(* If state methods are not disabled, run the stopped entry method. *)
IF NOT in_bDisableStateMethods THEN
	THIS^.M_LogMessage('Entered $'Stopped$' state.');
	THIS^.M110_Stopped_Entry();
ELSE
	THIS^.M_LogWarning('State methods disabled! Entered $'Stopped$' state. Waiting for transition...');
END_IF
END_ACTION

ACTION A111_Stopped:
{attribute 'hide'}
(* If state methods are not disabled, run the stopped method. *)
IF NOT in_bDisableStateMethods THEN
	THIS^.M111_Stopped(bReset => sm_bResetCmd, bAbort => sm_bAbortCmd);
	IF sm_bAbortCmd THEN
		sm_bAbort := TRUE;
	ELSIF sm_bResetCmd THEN
		sm_bReset := TRUE;
	END_IF
END_IF
END_ACTION

ACTION A112_Stopped_Exit:
{attribute 'hide'}
(* If state methods are not disabled, run the stopped exit method. *)
IF NOT in_bDisableStateMethods THEN
	THIS^.M112_Stopped_Exit();
END_IF
END_ACTION

{attribute 'hide'}
METHOD M110_Stopped_Entry : BOOL
END_METHOD

{attribute 'hide'}
METHOD M111_Stopped : BOOL
VAR_OUTPUT
	(* Move to the Resetting state*)
	bReset	: BOOL	:= FALSE;
	(* Move to the Aborting state*)
	bAbort	: BOOL	:= FALSE;
END_VAR
END_METHOD

{attribute 'hide'}
METHOD M112_Stopped_Exit : BOOL
END_METHOD

ACTION A200_Resetting_Entry:
{attribute 'hide'}
sm_enumState := E_PackMLState.Resetting;
sm_bIdle := FALSE;
sm_bStop := FALSE;

IF NOT in_bDisableStateMethods THEN
	THIS^.M_LogMessage('Entered $'Resetting$' state.');
	THIS^.M200_Resetting_Entry();
ELSE
	THIS^.M_LogWarning('State methods disabled! Entered $'Resetting$' state. Skipping to $'Idle$' state...');
	sm_bIdle := TRUE;
END_IF
END_ACTION

ACTION A201_Resetting:
{attribute 'hide'}
IF NOT in_bDisableStateMethods THEN
	THIS^.M201_Resetting(bIdle => sm_bIdleCmd, bStop => sm_bStopCmd, bAbort => sm_bAbortCmd);
	IF sm_bAbortCmd THEN
		sm_bAbort := TRUE;
	ELSIF sm_bStopCmd THEN
		sm_bStop := TRUE;
	ELSIF sm_bIdleCmd THEN
		sm_bIdle := TRUE;
	END_IF
END_IF
END_ACTION

ACTION A202_Resetting_Exit:
{attribute 'hide'}
IF NOT in_bDisableStateMethods THEN
	THIS^.M202_Resetting_Exit();
END_IF
END_ACTION

{attribute 'hide'}
METHOD M200_Resetting_Entry : BOOL
END_METHOD

{attribute 'hide'}
METHOD M201_Resetting : BOOL
VAR_OUTPUT
	(* Move to the Idle state*)
	bIdle	: BOOL	:= FALSE;
	(* Move to the Stopping state*)
	bStop	: BOOL	:= FALSE;
	(* Move to the Aborting state*)
	bAbort	: BOOL	:= FALSE;
END_VAR
// Move to idle state by default
bIdle := TRUE;
END_METHOD

{attribute 'hide'}
METHOD M202_Resetting_Exit : BOOL
END_METHOD

ACTION A210_Idle_Entry:
{attribute 'hide'}
sm_enumState := E_PackMLState.Idle;
sm_bStart := FALSE;

IF NOT in_bDisableStateMethods THEN
	THIS^.M_LogMessage('Entered $'Idle$' state.');
	THIS^.M210_Idle_Entry();
ELSE
	THIS^.M_LogWarning('State methods disabled! Entered $'Idle$' state. Waiting for transtion...');
END_IF
END_ACTION

ACTION A211_Idle:
{attribute 'hide'}
IF NOT in_bDisableStateMethods THEN
	THIS^.M211_Idle(bStart => sm_bStartCmd, bStop => sm_bStopCmd, bAbort => sm_bAbortCmd);
	IF sm_bAbortCmd THEN
		sm_bAbort := TRUE;
	ELSIF sm_bStopCmd THEN
		sm_bStop := TRUE;
	ELSIF sm_bStartCmd THEN
		sm_bStart := TRUE;
	END_IF
END_IF
END_ACTION

ACTION A212_Idle_Exit:
{attribute 'hide'}
IF NOT in_bDisableStateMethods THEN
	THIS^.M212_Idle_Exit();
END_IF
END_ACTION

{attribute 'hide'}
METHOD M210_Idle_Entry : BOOL
END_METHOD

{attribute 'hide'}
METHOD M211_Idle : BOOL
VAR_OUTPUT
	(* Move to the Starting state*)
	bStart	: BOOL	:= FALSE;
	(* Move to the Stopping state*)
	bStop	: BOOL	:= FALSE;
	(* Move to the Aborting state*)
	bAbort	: BOOL	:= FALSE;
END_VAR
END_METHOD

{attribute 'hide'}
METHOD M212_Idle_Exit : BOOL
END_METHOD

ACTION A300_Starting_Entry:
{attribute 'hide'}
sm_enumState := E_PackMLState.Starting;
sm_bStarted := FALSE;

IF NOT in_bDisableStateMethods THEN
	THIS^.M_LogMessage('Entered $'Starting$' state.');
	THIS^.M300_Starting_Entry();
ELSE
	THIS^.M_LogWarning('State methods disabled! Entered $'Starting$' state. Skipping to $'Execute$' state...');
	sm_bStarted := TRUE;
END_IF
END_ACTION

ACTION A301_Starting:
{attribute 'hide'}
IF NOT in_bDisableStateMethods THEN
	THIS^.M301_Starting(
		bStarted => sm_bStartedCmd,
		bStop => sm_bStopCmd,
		bAbort => sm_bAbortCmd);
	IF sm_bAbortCmd THEN
		sm_bAbort := TRUE;
	ELSIF sm_bStopCmd THEN
		sm_bStop := TRUE;
	ELSIF sm_bStartedCmd THEN
		sm_bStarted := TRUE;
	END_IF
END_IF
END_ACTION

ACTION A302_Starting_Exit:
{attribute 'hide'}
IF NOT in_bDisableStateMethods THEN
	THIS^.M302_Starting_Exit();
END_IF
END_ACTION

{attribute 'hide'}
METHOD M300_Starting_Entry : BOOL
END_METHOD

{attribute 'hide'}
METHOD M301_Starting : BOOL
VAR_OUTPUT
	(* Move to the Execute state*)
	bStarted	: BOOL	:= FALSE;
	(* Move to the Stopping state*)
	bStop		: BOOL	:= FALSE;
	(* Move to the Aborting state*)
	bAbort		: BOOL	:= FALSE;
END_VAR
// Move to execute state by default
bStarted := TRUE;
END_METHOD

{attribute 'hide'}
METHOD M302_Starting_Exit : BOOL
END_METHOD

ACTION A310_Execute_Entry:
{attribute 'hide'}
sm_enumState := E_PackMLState.Execute;
sm_bFinished := FALSE;
sm_bHold := FALSE;
sm_bSuspend := FALSE;

IF NOT in_bDisableStateMethods THEN
	THIS^.M_LogMessage('Entered $'Execute$' state.');
	THIS^.M310_Execute_Entry();
ELSE
	THIS^.M_LogWarning('State methods disabled! Entered $'Execute$' state. Waiting for transition...');
END_IF
END_ACTION

ACTION A311_Execute:
{attribute 'hide'}
IF NOT in_bDisableStateMethods THEN
	THIS^.M311_Execute(
		bFinished => sm_bFinishedCmd,
		bHold => sm_bHoldCmd,
		bSuspend => sm_bSuspendCmd,
		bStop => sm_bStopCmd,
		bAbort => sm_bAbortCmd);
	IF sm_bAbortCmd THEN
		sm_bAbort := TRUE;
	ELSIF sm_bStopCmd THEN
		sm_bStop := TRUE;
	ELSIF sm_bHoldCmd THEN
		sm_bHold := TRUE;
	ELSIF sm_bSuspendCmd THEN
		sm_bSuspend := TRUE;
	ELSIF sm_bFinishedCmd THEN
		sm_bFinished := TRUE;
	END_IF
END_IF
END_ACTION

ACTION A312_Execute_Exit:
{attribute 'hide'}
IF NOT in_bDisableStateMethods THEN
	THIS^.M312_Execute_Exit();
END_IF
END_ACTION

{attribute 'hide'}
METHOD M310_Execute_Entry : BOOL
END_METHOD

{attribute 'hide'}
METHOD M311_Execute : BOOL
VAR_OUTPUT
	(* Move to the Completing state*)
	bFinished	: BOOL	:= FALSE;
	(* Move to the Holding state*)
	bHold		: BOOL	:= FALSE;
	(* Move to the Suspending state*)
	bSuspend	: BOOL	:= FALSE;
	(* Move to the Stopping state*)
	bStop		: BOOL	:= FALSE;
	(* Move to the Aborting state*)
	bAbort		: BOOL	:= FALSE;
END_VAR
END_METHOD

{attribute 'hide'}
METHOD M312_Execute_Exit : BOOL
END_METHOD

ACTION A320_Completing_Entry:
{attribute 'hide'}
sm_enumState := E_PackMLState.Completing;
sm_bCompleted := FALSE;

IF NOT in_bDisableStateMethods THEN
	THIS^.M_LogMessage('Entered $'Completing$' state.');
	THIS^.M320_Completing_Entry();
ELSE
	THIS^.M_LogWarning('State methods disabled! Entered $'Completing$' state. Skipping to $'Completed$' state...');
	sm_bCompleted := TRUE;
END_IF
END_ACTION

ACTION A321_Completing:
{attribute 'hide'}
IF NOT in_bDisableStateMethods THEN
	THIS^.M321_Completing(
		bCompleted => sm_bCompletedCmd,
		bStop => sm_bStopCmd,
		bAbort => sm_bAbortCmd);
	IF sm_bAbortCmd THEN
		sm_bAbort := TRUE;
	ELSIF sm_bStopCmd THEN
		sm_bStop := TRUE;
	ELSIF sm_bCompletedCmd THEN
		sm_bCompleted := TRUE;
	END_IF
END_IF
END_ACTION

ACTION A322_Completing_Exit:
{attribute 'hide'}
IF NOT in_bDisableStateMethods THEN
	THIS^.M322_Completing_Exit();
END_IF
END_ACTION

{attribute 'hide'}
METHOD M320_Completing_Entry : BOOL
END_METHOD

{attribute 'hide'}
METHOD M321_Completing : BOOL
VAR_OUTPUT
	(* Move to the Complete state*)
	bCompleted	: BOOL	:= FALSE;
	(* Move to the Stopping state*)
	bStop		: BOOL	:= FALSE;
	(* Move to the Aborting state*)
	bAbort		: BOOL	:= FALSE;
END_VAR
// Move to complete state by default.
bCompleted := TRUE;
END_METHOD

{attribute 'hide'}
METHOD M322_Completing_Exit : BOOL
END_METHOD

ACTION A330_Complete_Entry:
{attribute 'hide'}
sm_enumState := E_PackMLState.Complete;
sm_bReturn := FALSE;

IF NOT in_bDisableStateMethods THEN
	THIS^.M_LogMessage('Entered $'Complete$' state.');
	THIS^.M330_Complete_Entry();
ELSE
	THIS^.M_LogWarning('State methods disabled! Entered $'Complete$' state. Waiting for transition...');
END_IF
END_ACTION

ACTION A331_Complete:
{attribute 'hide'}
IF NOT in_bDisableStateMethods THEN
	THIS^.M331_Complete(
		bReturn => sm_bReturnCmd,
		bStop => sm_bStopCmd,
		bAbort => sm_bAbortCmd);
	IF sm_bAbortCmd THEN
		sm_bAbort := TRUE;
	ELSIF sm_bStopCmd THEN
		sm_bStop := TRUE;
	ELSIF sm_bReturnCmd THEN
		sm_bReturn := TRUE;
	END_IF
END_IF
END_ACTION

ACTION A332_Complete_Exit:
{attribute 'hide'}
IF NOT in_bDisableStateMethods THEN
	THIS^.M332_Complete_Exit();
END_IF
END_ACTION

{attribute 'hide'}
METHOD M330_Complete_Entry : BOOL
END_METHOD

{attribute 'hide'}
METHOD M331_Complete : BOOL
VAR_OUTPUT
	(* Move to the Resetting state*)
	bReturn	: BOOL	:= FALSE;
	(* Move to the Stopping state*)
	bStop	: BOOL	:= FALSE;
	(* Move to the Aborting state*)
	bAbort	: BOOL	:= FALSE;
END_VAR
END_METHOD

{attribute 'hide'}
METHOD M332_Complete_Exit : BOOL
END_METHOD

ACTION A400_Holding_Entry:
{attribute 'hide'}
sm_enumState := E_PackMLState.Holding;
sm_bHeld := FALSE;

IF NOT in_bDisableStateMethods THEN
	THIS^.M_LogMessage('Entered $'Holding$' state.');
	THIS^.M400_Holding_Entry();
ELSE
	THIS^.M_LogMessage('State methods disabled! Entered $'Holding$' state. Skipping to $'Held$' state...');
	sm_bHeld := TRUE;
END_IF
END_ACTION

ACTION A401_Holding:
{attribute 'hide'}
IF NOT in_bDisableStateMethods THEN
	THIS^.M401_Holding(
		bHeld => sm_bHeldCmd,
		bStop => sm_bStopCmd,
		bAbort => sm_bAbortCmd);
	IF sm_bAbortCmd THEN
		sm_bAbort := TRUE;
	ELSIF sm_bStopCmd THEN
		sm_bStop := TRUE;
	ELSIF sm_bHeldCmd THEN
		sm_bHeld := TRUE;
	END_IF
END_IF
END_ACTION

ACTION A402_Holding_Exit:
{attribute 'hide'}
IF NOT in_bDisableStateMethods THEN
	THIS^.M402_Holding_Exit();
END_IF
END_ACTION

{attribute 'hide'}
METHOD M400_Holding_Entry : BOOL
END_METHOD

{attribute 'hide'}
METHOD M401_Holding : BOOL
VAR_OUTPUT
	(* Move to the Held state*)
	bHeld	: BOOL	:= FALSE;
	(* Move to the Stopping state*)
	bStop	: BOOL	:= FALSE;
	(* Move to the Aborting state*)
	bAbort	: BOOL	:= FALSE;
END_VAR
// Move to held state by default
bHeld := TRUE;
END_METHOD

{attribute 'hide'}
METHOD M402_Holding_Exit : BOOL
END_METHOD

ACTION A410_Held_Entry:
{attribute 'hide'}
sm_enumState := E_PackMLState.Held;
sm_bUnhold := FALSE;

IF NOT in_bDisableStateMethods THEN
	THIS^.M_LogMessage('Entered $'Held$' state.');
	THIS^.M410_Held_Entry();
ELSE
	THIS^.M_LogWarning('State methods disabled! Entered $'Held$' state. Waiting for transition...');
END_IF
END_ACTION

ACTION A411_Held:
{attribute 'hide'}
IF NOT in_bDisableStateMethods THEN
	THIS^.M411_Held(
		bUnhold => sm_bUnholdCmd,
		bStop => sm_bStopCmd,
		bAbort => sm_bAbortCmd);
	IF sm_bAbortCmd THEN
		sm_bAbort := TRUE;
	ELSIF sm_bStopCmd THEN
		sm_bStop := TRUE;
	ELSIF sm_bUnholdCmd THEN
		sm_bUnhold := TRUE;
	END_IF
END_IF
END_ACTION

ACTION A412_Held_Exit:
{attribute 'hide'}
IF NOT in_bDisableStateMethods THEN
	THIS^.M412_Held_Exit();
END_IF
END_ACTION

{attribute 'hide'}
METHOD M410_Held_Entry : BOOL
END_METHOD

{attribute 'hide'}
METHOD M411_Held : BOOL
VAR_OUTPUT
	(* Move to the Unholding state*)
	bUnhold	: BOOL	:= FALSE;
	(* Move to the Stopping state*)
	bStop	: BOOL	:= FALSE;
	(* Move to the Aborting state*)
	bAbort	: BOOL	:= FALSE;
END_VAR
END_METHOD

{attribute 'hide'}
METHOD M412_Held_Exit : BOOL
END_METHOD

ACTION A420_Unholding_Entry:
{attribute 'hide'}
sm_enumState := E_PackMLState.Unholding;
sm_bUnheld := FALSE;

IF NOT in_bDisableStateMethods THEN
	THIS^.M_LogMessage('Entered $'Unholding$' state.');
	THIS^.M420_Unholding_Entry();
ELSE
	THIS^.M_LogMessage('State methods disabled! Entered $'Unholding$' state. Skipping to $'Execute$' state.');
	sm_bUnheld := TRUE;
END_IF
END_ACTION

ACTION A421_Unholding:
{attribute 'hide'}
IF NOT in_bDisableStateMethods THEN
	THIS^.M421_Unholding(
		bUnheld => sm_bUnheldCmd,
		bStop => sm_bStopCmd,
		bAbort => sm_bAbortCmd);
	IF sm_bAbortCmd THEN
		sm_bAbort := TRUE;
	ELSIF sm_bStopCmd THEN
		sm_bStop := TRUE;
	ELSIF sm_bUnheldCmd THEN
		sm_bUnheld := TRUE;
	END_IF
END_IF
END_ACTION

ACTION A422_Unholding_Exit:
{attribute 'hide'}
IF NOT in_bDisableStateMethods THEN
	THIS^.M422_Unholding_Exit();
END_IF
END_ACTION

{attribute 'hide'}
METHOD M420_Unholding_Entry : BOOL
END_METHOD

{attribute 'hide'}
METHOD M421_Unholding : BOOL
VAR_OUTPUT
	(* Move to the Execute state*)
	bUnheld	: BOOL	:= FALSE;
	(* Move to the Stopping state*)
	bStop	: BOOL	:= FALSE;
	(* Move to the Aborting state*)
	bAbort	: BOOL	:= FALSE;
END_VAR
// Move to execute state by default
bUnheld := TRUE;
END_METHOD

{attribute 'hide'}
METHOD M422_Unholding_Exit : BOOL
END_METHOD

ACTION A500_Suspending_Entry:
{attribute 'hide'}
sm_enumState := E_PackMLState.Suspending;
sm_bSuspended := FALSE;

IF NOT in_bDisableStateMethods THEN
	THIS^.M_LogMessage('Entered $'Suspending$' state.');
	THIS^.M500_Suspending_Entry();
ELSE
	THIS^.M_LogWarning('State methods disabled! Entered $'Suspending$' state. Skipping to $'Suspended$' state...');
	sm_bSuspended := TRUE;
END_IF
END_ACTION

ACTION A501_Suspending:
{attribute 'hide'}
IF NOT in_bDisableStateMethods THEN
	THIS^.M501_Suspending(
		bSuspended => sm_bSuspendedCmd,
		bStop => sm_bStopCmd,
		bAbort => sm_bAbortCmd);
	IF sm_bAbortCmd THEN
		sm_bAbort := TRUE;
	ELSIF sm_bStopCmd THEN
		sm_bStop := TRUE;
	ELSIF sm_bSuspendedCmd THEN
		sm_bSuspended := TRUE;
	END_IF
END_IF
END_ACTION

ACTION A502_Suspending_Exit:
{attribute 'hide'}
IF NOT in_bDisableStateMethods THEN
	THIS^.M502_Suspending_Exit();
END_IF
END_ACTION

{attribute 'hide'}
METHOD M500_Suspending_Entry : BOOL
END_METHOD

{attribute 'hide'}
METHOD M501_Suspending : BOOL
VAR_OUTPUT
	(* Move to the Suspended state*)
	bSuspended	: BOOL	:= FALSE;
	(* Move to the Stopping state*)
	bStop		: BOOL	:= FALSE;
	(* Move to the Aborting state*)
	bAbort		: BOOL	:= FALSE;
END_VAR
// Go to suspended state by default
bSuspended := TRUE;
END_METHOD

{attribute 'hide'}
METHOD M502_Suspending_Exit : BOOL
END_METHOD

ACTION A510_Suspended_Entry:
{attribute 'hide'}
sm_enumState := E_PackMLState.Suspended;
sm_bUnsuspend := FALSE;

IF NOT in_bDisableStateMethods THEN
	THIS^.M_LogMessage('Entered $'Suspended$' state.');
	THIS^.M510_Suspended_Entry();
ELSE
	THIS^.M_LogWarning('State methods disabled! Entered $'Suspended$' state. Waiting for transition...');
END_IF
END_ACTION

ACTION A511_Suspended:
{attribute 'hide'}
IF NOT in_bDisableStateMethods THEN
	THIS^.M511_Suspended(
		bUnsuspend => sm_bUnsuspendCmd,
		bStop => sm_bStopCmd,
		bAbort => sm_bAbortCmd);
	IF sm_bAbortCmd THEN
		sm_bAbort := TRUE;
	ELSIF sm_bStopCmd THEN
		sm_bStop := TRUE;
	ELSIF sm_bUnsuspendCmd THEN
		sm_bUnsuspend := TRUE;
	END_IF
END_IF
END_ACTION

ACTION A512_Suspended_Exit:
{attribute 'hide'}
IF NOT in_bDisableStateMethods THEN
	THIS^.M512_Suspended_Exit();
END_IF
END_ACTION

{attribute 'hide'}
METHOD M510_Suspended_Entry : BOOL
END_METHOD

{attribute 'hide'}
METHOD M511_Suspended : BOOL
VAR_OUTPUT
	(* Move to the Unsuspending state*)
	bUnsuspend	: BOOL	:= FALSE;
	(* Move to the Stopping state*)
	bStop		: BOOL	:= FALSE;
	(* Move to the Aborting state*)
	bAbort		: BOOL	:= FALSE;
END_VAR
END_METHOD

{attribute 'hide'}
METHOD M512_Suspended_Exit : BOOL
END_METHOD

ACTION A520_Unsuspending_Entry:
{attribute 'hide'}
sm_enumState := E_PackMLState.Unsuspending;
sm_bUnsuspended := FALSE;

IF NOT in_bDisableStateMethods THEN
	THIS^.M_LogMessage('Entered $'Unsuspending$' state.');
	THIS^.M520_Unsuspending_Entry();
ELSE
	THIS^.M_LogWarning('State methods disabled! Entered $'Unsuspending$' state. Skipping to $'Execute$' state...');
	sm_bUnsuspended := TRUE;
END_IF
END_ACTION

ACTION A521_Unsuspending:
{attribute 'hide'}
IF NOT in_bDisableStateMethods THEN
	THIS^.M521_Unsuspending(
		bUnsuspended => sm_bUnsuspendedCmd,
		bStop => sm_bStopCmd,
		bAbort => sm_bAbortCmd);
	IF sm_bAbortCmd THEN
		sm_bAbort := TRUE;
	ELSIF sm_bStopCmd THEN
		sm_bStop := TRUE;
	ELSIF sm_bUnsuspendedCmd THEN
		sm_bUnsuspended := TRUE;
	END_IF
END_IF
END_ACTION

ACTION A522_Unsuspending_Exit:
{attribute 'hide'}
IF NOT in_bDisableStateMethods THEN
	THIS^.M522_Unsuspending_Exit();
END_IF
END_ACTION

{attribute 'hide'}
METHOD M520_Unsuspending_Entry : BOOL
END_METHOD

{attribute 'hide'}
METHOD M521_Unsuspending : BOOL
VAR_OUTPUT
	(* Move to the Execute state*)
	bUnsuspended	: BOOL	:= FALSE;
	(* Move to the Stopping state*)
	bStop			: BOOL	:= FALSE;
	(* Move to the Aborting state*)
	bAbort			: BOOL	:= FALSE;
END_VAR
// Move to the execute state by default
bUnsuspended := TRUE;
END_METHOD

{attribute 'hide'}
METHOD M522_Unsuspending_Exit : BOOL
END_METHOD

ACTION A_StateMachine:
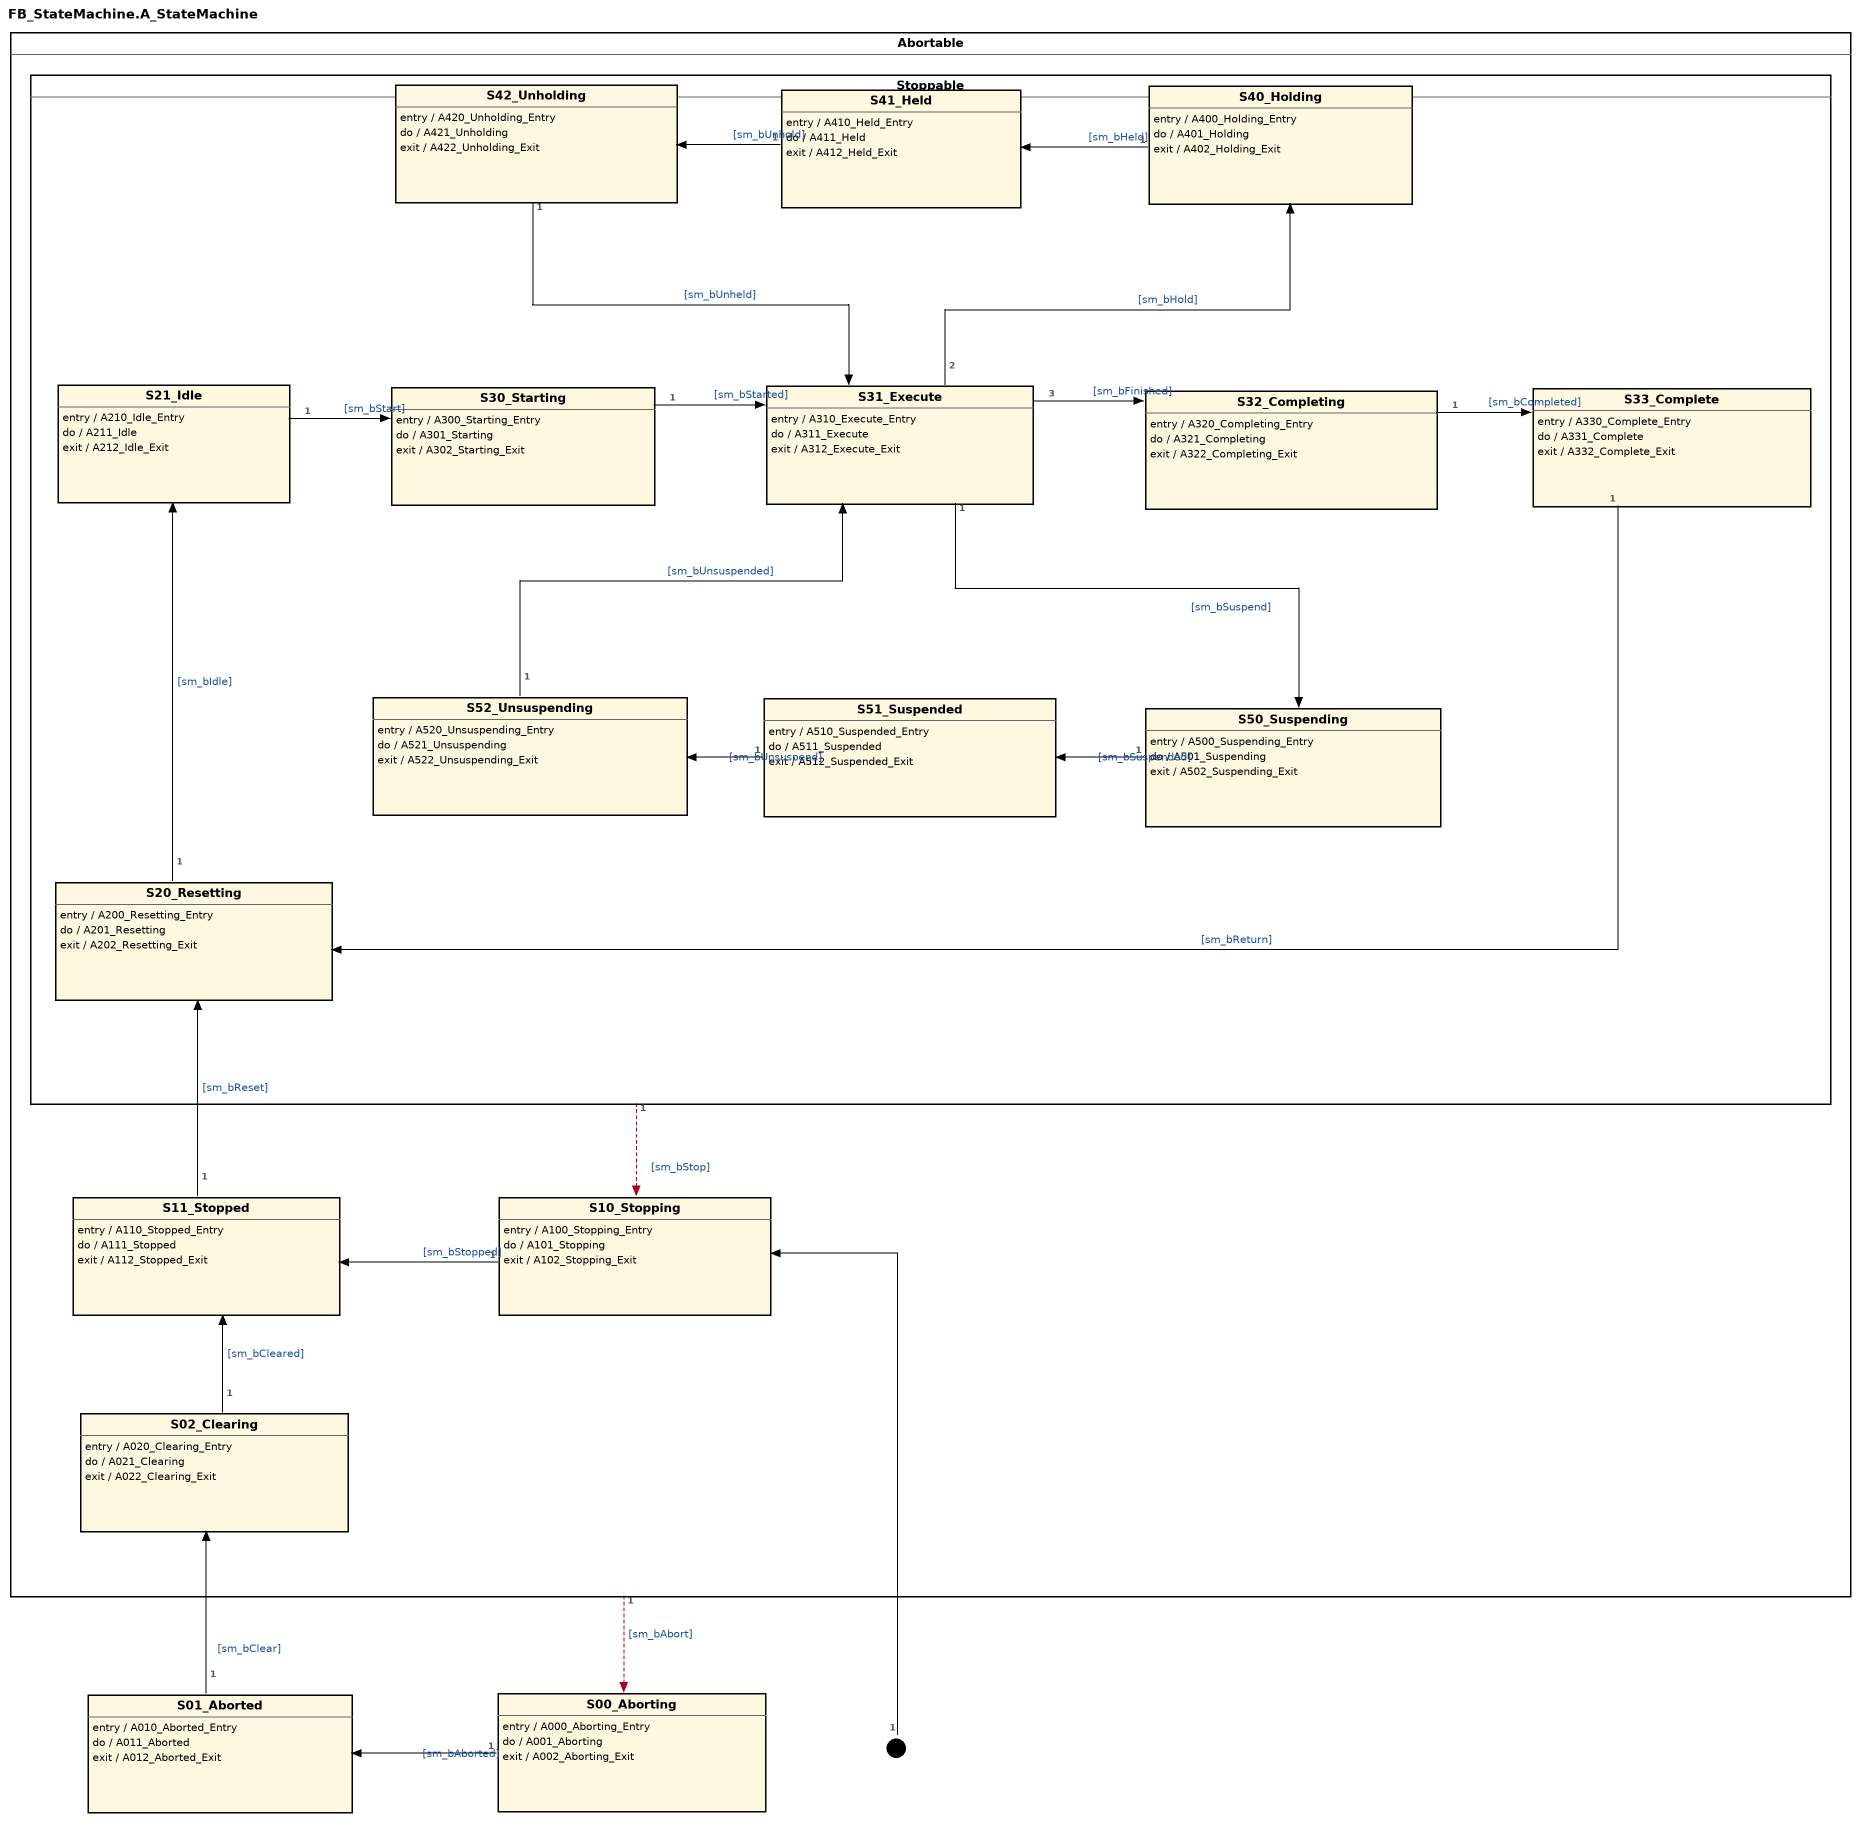
STATECHART A_StateMachine  // abortable
    START StartState1
    COMPOSITE STATE Abortable
        COMPOSITE STATE Stoppable
            STATE S42_Unholding
                entry / A420_Unholding_Entry
                do / A421_Unholding
                exit / A422_Unholding_Exit
            STATE S41_Held
                entry / A410_Held_Entry
                do / A411_Held
                exit / A412_Held_Exit
            STATE S40_Holding
                entry / A400_Holding_Entry
                do / A401_Holding
                exit / A402_Holding_Exit
            STATE S21_Idle
                entry / A210_Idle_Entry
                do / A211_Idle
                exit / A212_Idle_Exit
            STATE S30_Starting
                entry / A300_Starting_Entry
                do / A301_Starting
                exit / A302_Starting_Exit
            STATE S31_Execute
                entry / A310_Execute_Entry
                do / A311_Execute
                exit / A312_Execute_Exit
            STATE S32_Completing
                entry / A320_Completing_Entry
                do / A321_Completing
                exit / A322_Completing_Exit
            STATE S33_Complete
                entry / A330_Complete_Entry
                do / A331_Complete
                exit / A332_Complete_Exit
            STATE S52_Unsuspending
                entry / A520_Unsuspending_Entry
                do / A521_Unsuspending
                exit / A522_Unsuspending_Exit
            STATE S51_Suspended
                entry / A510_Suspended_Entry
                do / A511_Suspended
                exit / A512_Suspended_Exit
            STATE S50_Suspending
                entry / A500_Suspending_Entry
                do / A501_Suspending
                exit / A502_Suspending_Exit
            STATE S20_Resetting
                entry / A200_Resetting_Entry
                do / A201_Resetting
                exit / A202_Resetting_Exit
            S42_Unholding -> S31_Execute [sm_bUnheld] // priority 1
            S41_Held -> S42_Unholding [sm_bUnhold] // priority 1
            S40_Holding -> S41_Held [sm_bHeld] // priority 1
            S21_Idle -> S30_Starting [sm_bStart] // priority 1
            S30_Starting -> S31_Execute [sm_bStarted] // priority 1
            S31_Execute -> S50_Suspending [sm_bSuspend] // priority 1
            S31_Execute -> S40_Holding [sm_bHold] // priority 2
            S31_Execute -> S32_Completing [sm_bFinished] // priority 3
            S32_Completing -> S33_Complete [sm_bCompleted] // priority 1
            S33_Complete -> S20_Resetting [sm_bReturn] // priority 1
            S52_Unsuspending -> S31_Execute [sm_bUnsuspended] // priority 1
            S51_Suspended -> S52_Unsuspending [sm_bUnsuspend] // priority 1
            S50_Suspending -> S51_Suspended [sm_bSuspended] // priority 1
            S20_Resetting -> S21_Idle [sm_bIdle] // priority 1
        END_STATE
        STATE S11_Stopped
            entry / A110_Stopped_Entry
            do / A111_Stopped
            exit / A112_Stopped_Exit
        STATE S10_Stopping
            entry / A100_Stopping_Entry
            do / A101_Stopping
            exit / A102_Stopping_Exit
        STATE S02_Clearing
            entry / A020_Clearing_Entry
            do / A021_Clearing
            exit / A022_Clearing_Exit
        Stoppable -> S10_Stopping [sm_bStop] // priority 1, exception
        S11_Stopped -> S20_Resetting [sm_bReset] // priority 1
        S10_Stopping -> S11_Stopped [sm_bStopped] // priority 1
        S02_Clearing -> S11_Stopped [sm_bCleared] // priority 1
    END_STATE
    STATE S01_Aborted
        entry / A010_Aborted_Entry
        do / A011_Aborted
        exit / A012_Aborted_Exit
    STATE S00_Aborting
        entry / A000_Aborting_Entry
        do / A001_Aborting
        exit / A002_Aborting_Exit
    StartState1 -> S10_Stopping  // priority 1, on completion
    Abortable -> S00_Aborting [sm_bAbort] // priority 1, exception
    S01_Aborted -> S02_Clearing [sm_bClear] // priority 1
    S00_Aborting -> S01_Aborted [sm_bAborted] // priority 1
END_STATECHART
END_ACTION

END_FUNCTION_BLOCK

// Interfaces/State Machine/I_StateControl
(* The state control interface should be implemented on stateful modules that
cannot move on from wait states automatically due to being controlled by
external modules. *)
INTERFACE I_StateControl

(* Go to the aborting state while in the stoppable or abortable group. *)
METHOD M_Abort : BOOL
VAR_INPUT
END_VAR
END_METHOD

(* Go to the clearing state from the aborted state. *)
METHOD M_Clear : BOOL
VAR_INPUT
END_VAR
END_METHOD

(* Go to the completing state from the execute state. *)
METHOD M_Complete : BOOL
VAR_INPUT
END_VAR
END_METHOD

(* Go to the holding state from the execute state. *)
METHOD M_Hold : BOOL
VAR_INPUT
END_VAR
END_METHOD

(* Go to the resetting state from the stopped state. *)
METHOD M_Reset : BOOL
VAR_INPUT
END_VAR
END_METHOD

(* Go to the execute state from the idle state. *)
METHOD M_Start : BOOL
VAR_INPUT
END_VAR
END_METHOD

(* Go to the stopping state while in the stoppable group. *)
METHOD M_Stop : BOOL
VAR_INPUT
END_VAR
END_METHOD

(* Go to the suspending state from the execute state. *)
METHOD M_Suspend : BOOL
VAR_INPUT
END_VAR
END_METHOD

(* Go to the unholding state from the held state. *)
METHOD M_Unhold : BOOL
VAR_INPUT
END_VAR
END_METHOD

(* Go to the unsuspending state from the suspended state. *)
METHOD M_Unsuspend : BOOL
VAR_INPUT
END_VAR
END_METHOD

END_INTERFACE

// Interfaces/Machines/I_MachineStationStateControl
INTERFACE I_MachineStationStateControl

(* Executes M_Abort on all stations and returns TRUE when M_Abort
	returns TRUE on all stations. *)
METHOD M_AbortStations : BOOL
VAR_INPUT
END_VAR
END_METHOD

(* Executes M_Clear on all stations and returns TRUE when M_Clear
	returns TRUE on all stations. *)
METHOD M_ClearStations : BOOL
VAR_INPUT
END_VAR
END_METHOD

(* Executes M_Complete on all stations and returns TRUE when M_Complete
	returns TRUE on all stations. *)
METHOD M_CompleteStations : BOOL
VAR_INPUT
END_VAR
END_METHOD

(* Executes M_Hold on all stations and returns TRUE when M_Hold 
	returns TRUE on all stations. *)
METHOD M_HoldStations : BOOL
VAR_INPUT
END_VAR
END_METHOD

(* Executes M_Reset on all stations and returns TRUE when M_Reset 
	returns TRUE on all stations. *)
METHOD M_ResetStations : BOOL
VAR_INPUT
END_VAR
END_METHOD

(* Executes M_Start on all stations and returns TRUE when M_Start 
	returns TRUE on all stations. *)
METHOD M_StartStations : BOOL
VAR_INPUT
END_VAR
END_METHOD

(* Executes M_Stop on all stations and returns TRUE when M_Stop 
	returns TRUE on all stations. *)
METHOD M_StopStations : BOOL
VAR_INPUT
END_VAR
END_METHOD

(* Executes M_Suspend on all stations and returns TRUE when M_Suspend
	returns TRUE on all stations. *)
METHOD M_SuspendStations : BOOL
VAR_INPUT
END_VAR
END_METHOD

(* Executes M_Unhold on all stations and returns TRUE when M_Unhold
	returns TRUE on all stations. *)
METHOD M_UnholdStations : BOOL
VAR_INPUT
END_VAR
END_METHOD

(* Executes M_Unsuspend on all stations and returns TRUE when M_Unsuspend
	returns TRUE on all stations. *)
METHOD M_UnsuspendStations : BOOL
VAR_INPUT
END_VAR
END_METHOD

END_INTERFACE

// Abstract/FB_Station
(*
===============================================================================
Station
===============================================================================
:Contact: Kevin Sanita <ksanita@sensata.com>
:Last Edited: March 2022

:Description: Represents a station, which is a collection of devices that interact with each other.

:Notes:
* Stations are able to implement state machines. To implement a state machine, implement I_Stateful
* In order for a state machine to run, THIS^.A_StateMachine must be called in the function block body.

:Change Log:
- **December 2021** Initial version
- **March 16, 2022** Added device list controls
*)
FUNCTION_BLOCK PUBLIC ABSTRACT FB_Station EXTENDS FB_StateMachine
	IMPLEMENTS I_SimpleTransitionStatesOnly // Has some basic default implementations
VAR_INPUT
END_VAR
VAR_OUTPUT
END_VAR
VAR
	sta_arrDevices : T_StationDeviceArray;
	
	sta_intAbortDevicesStep: INT;
	sta_intClearDevicesStep: INT;
	sta_intCompleteDevicesStep: INT;
	sta_intHoldDevicesStep: INT;
	sta_intResetDevicesStep: INT;
	sta_intStartDevicesStep: INT;
	sta_intStopDevicesStep: INT;
	sta_intSuspendDevicesStep: INT;
	sta_intUnholdDevicesStep: INT;
	sta_intUnsuspendDevicesStep: INT;
	
	sta_intAbortingStep: INT;
	sta_intClearingStep: INT;
	sta_intResettingStep: INT;
	sta_intStartingStep: INT;
	sta_intCompletingStep: INT;
	sta_intHoldingStep: INT;
	sta_intUnholdingStep: INT;
	sta_intSuspendingStep: INT;
	sta_intUnsuspendingStep: INT;
	sta_intStoppingStep: INT;
END_VAR

(* The 'Aborting' state can be entered at any time while within the 'abortable'
section of the state machine. It is typically entered in response to an 'Abort'
command or a critical fault. The logic should safely but rapidly bring the
components of the module to a stop while maintaining as much information about
the pre-abort scenario as possible. *)
METHOD M001_Aborting : BOOL
VAR_OUTPUT
	(* This should be set to true once all components of the module have safely
	come to a stop. Once set to true, the state machine will move to the
	'Aborted' state. *)
	bAborted	: BOOL;
END_VAR
VAR
	_bStepComplete: BOOL;
	_intStep: INT;
END_VAR
VAR_INST // added by the converter: edge detectors and wires of the graphical bodies
    _w1, _w2, _w3 : BOOL;
END_VAR
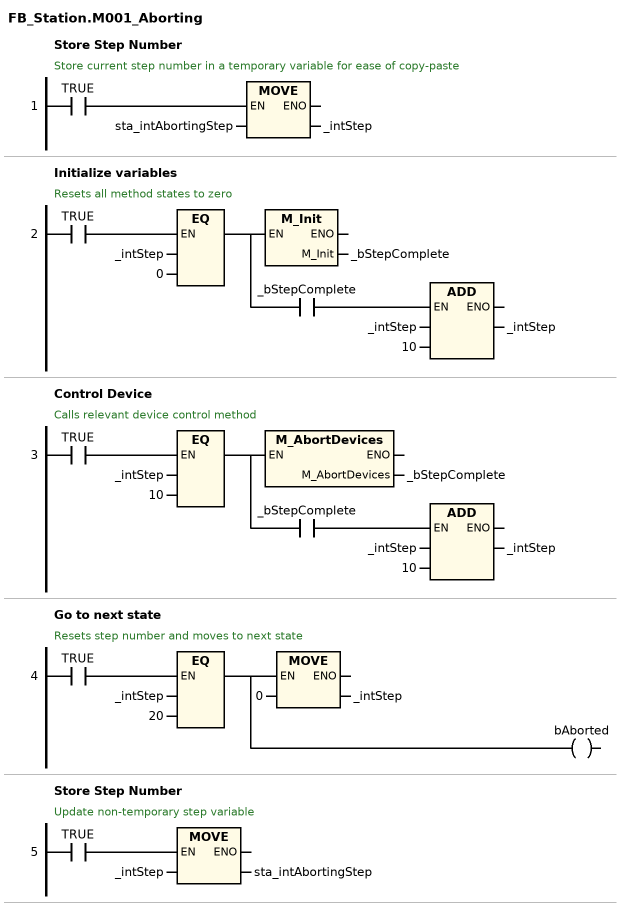
// NETWORK 1: Store Step Number
// Store current step number in a temporary variable for ease of copy-paste
_intStep := sta_intAbortingStep;

// NETWORK 2: Initialize variables
// Resets all method states to zero
_w1 := _intStep = 0;
IF _w1 THEN _bStepComplete := M_Init(); END_IF
IF _w1 AND _bStepComplete THEN _intStep := _intStep + 10; END_IF

// NETWORK 3: Control Device
// Calls relevant device control method
_w2 := _intStep = 10;
IF _w2 THEN _bStepComplete := M_AbortDevices(); END_IF
IF _w2 AND _bStepComplete THEN _intStep := _intStep + 10; END_IF

// NETWORK 4: Go to next state
// Resets step number and moves to next state
_w3 := _intStep = 20;
IF _w3 THEN _intStep := 0; END_IF
bAborted := _w3;

// NETWORK 5: Store Step Number
// Update non-temporary step variable
sta_intAbortingStep := _intStep;
END_METHOD

(* This state should clear any faults and reset any safety features related
to the module, as well as perform actions similar to the 'Stopping' state
if they were not already performed while aborting. *)
METHOD M021_Clearing : BOOL
VAR_OUTPUT
	(* This should be set to true once the safety state of all module
	components are reset and all errors are cleared. *)
	bCleared	: BOOL;
	(* This should be set to true if a potentially hazardous error or a safety
	fault has occurred in any tasks. Once set to true, the state machine will
	move to the 'Aborting' state. *)
	bAbort	: BOOL;
END_VAR
VAR
	_bStepComplete: BOOL;
	_intStep: INT;
END_VAR
VAR_INST // added by the converter: edge detectors and wires of the graphical bodies
    _w1, _w2, _w3, _w4, _w5 : BOOL;
END_VAR
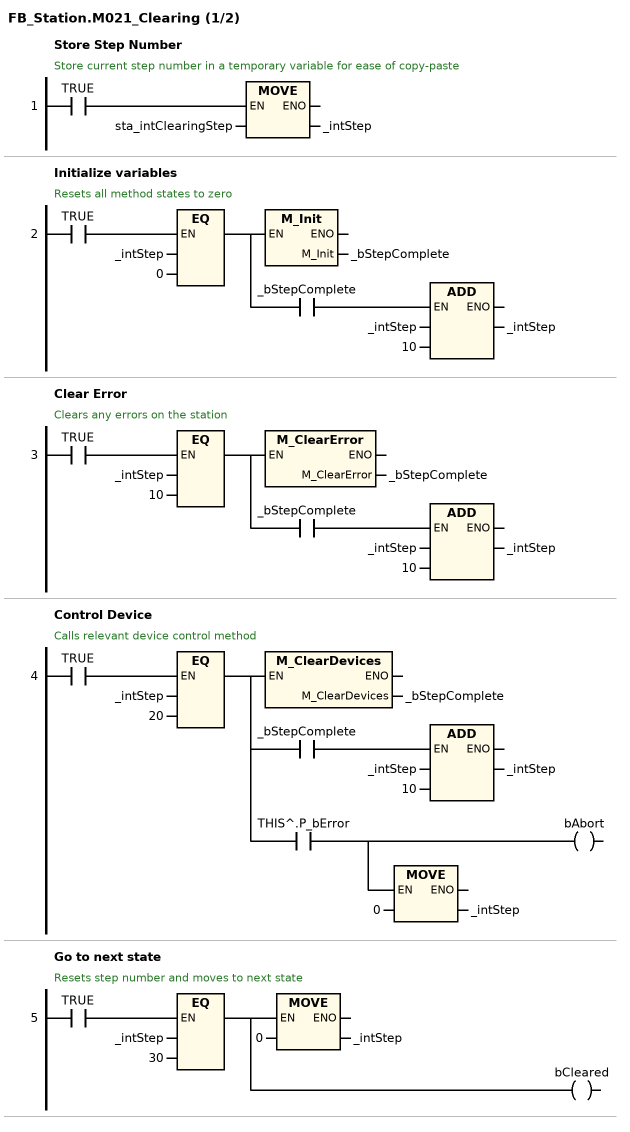
// NETWORK 1: Store Step Number
// Store current step number in a temporary variable for ease of copy-paste
_intStep := sta_intClearingStep;

// NETWORK 2: Initialize variables
// Resets all method states to zero
_w1 := _intStep = 0;
IF _w1 THEN _bStepComplete := M_Init(); END_IF
IF _w1 AND _bStepComplete THEN _intStep := _intStep + 10; END_IF

// NETWORK 3: Clear Error
// Clears any errors on the station
_w2 := _intStep = 10;
IF _w2 THEN _bStepComplete := M_ClearError(); END_IF
IF _w2 AND _bStepComplete THEN _intStep := _intStep + 10; END_IF

// NETWORK 4: Control Device
// Calls relevant device control method
_w3 := _intStep = 20;
IF _w3 THEN _bStepComplete := M_ClearDevices(); END_IF
IF _w3 AND _bStepComplete THEN _intStep := _intStep + 10; END_IF
_w4 := _w3 AND THIS^.P_bError;
bAbort := _w4;
IF _w4 THEN _intStep := 0; END_IF

// NETWORK 5: Go to next state
// Resets step number and moves to next state
_w5 := _intStep = 30;
IF _w5 THEN _intStep := 0; END_IF
bCleared := _w5;

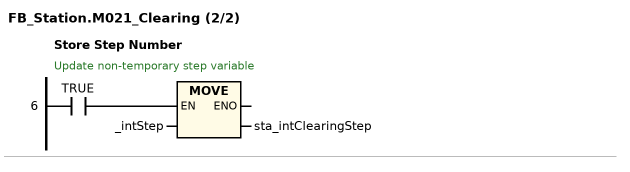
// NETWORK 6: Store Step Number
// Update non-temporary step variable
sta_intClearingStep := _intStep;
END_METHOD

(* This state can be entered from anywhere within the 'stoppable' group of
states. This state should safely bring the components of the module to a
controlled stop and then move to the 'Stopped' state once completed. *)
METHOD M101_Stopping : BOOL
VAR_OUTPUT
	(* This should be set to true once all relevant components have come to a
	controlled stop. Once set to true, the state machine will move to the
	'Stopped' state. *)
	bStopped	: BOOL;
	(* This should be set to true if a potentially hazardous error or a safety
	fault has occurred in any tasks. Once set to true, the state machine will
	move to the 'Aborting' state. *)
	bAbort	: BOOL;
END_VAR
VAR
	_bStepComplete: BOOL;
	_intStep: INT;
	sta_intStartingStep: INT;
END_VAR
VAR_INST // added by the converter: edge detectors and wires of the graphical bodies
    _w1, _w2, _w3, _w4 : BOOL;
END_VAR
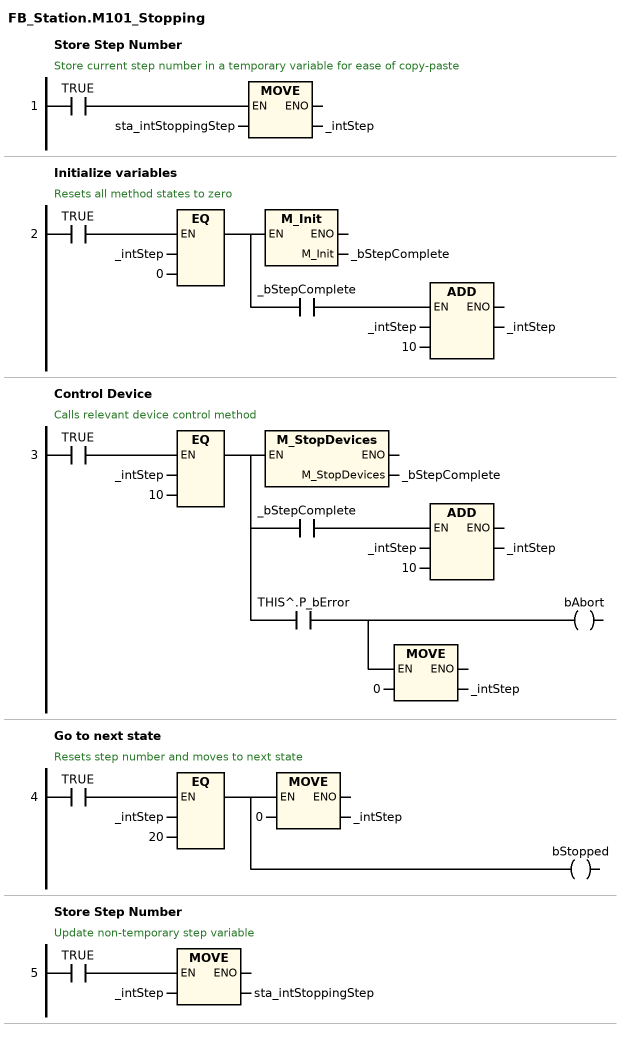
// NETWORK 1: Store Step Number
// Store current step number in a temporary variable for ease of copy-paste
_intStep := sta_intStoppingStep;

// NETWORK 2: Initialize variables
// Resets all method states to zero
_w1 := _intStep = 0;
IF _w1 THEN _bStepComplete := M_Init(); END_IF
IF _w1 AND _bStepComplete THEN _intStep := _intStep + 10; END_IF

// NETWORK 3: Control Device
// Calls relevant device control method
_w2 := _intStep = 10;
IF _w2 THEN _bStepComplete := M_StopDevices(); END_IF
IF _w2 AND _bStepComplete THEN _intStep := _intStep + 10; END_IF
_w3 := _w2 AND THIS^.P_bError;
bAbort := _w3;
IF _w3 THEN _intStep := 0; END_IF

// NETWORK 4: Go to next state
// Resets step number and moves to next state
_w4 := _intStep = 20;
IF _w4 THEN _intStep := 0; END_IF
bStopped := _w4;

// NETWORK 5: Store Step Number
// Update non-temporary step variable
sta_intStoppingStep := _intStep;
END_METHOD

(* This state should place the module and all of its components into a safe
energized idle state where it will wait for a start command. Once all tasks are
complete, it will move to the 'Idle' state. No external movement should occur
as a result of this state. *)
METHOD M201_Resetting : BOOL
VAR_OUTPUT
	(* Set this to true once the module is energized and ready to start.
	Once set to true, the state machine will move to the 'Idle' state. *)
	bIdle	: BOOL;
	(* This should be set to true if an external source requests that the module
	exit its current state and come to a controlled stop. Once set to true, the
	state machine will move to the 'Stopping' state. *)
	bStop	: BOOL;
	(* This should be set to true if a potentially hazardous error or a safety
	fault has occurred in any tasks. Once set to true, the state machine will
	move to the 'Aborting' state. *)
	bAbort	: BOOL;
END_VAR
VAR
	_bStepComplete: BOOL;
	_intStep: INT;
END_VAR
VAR_INST // added by the converter: edge detectors and wires of the graphical bodies
    _w1, _w2, _w3, _w4 : BOOL;
END_VAR
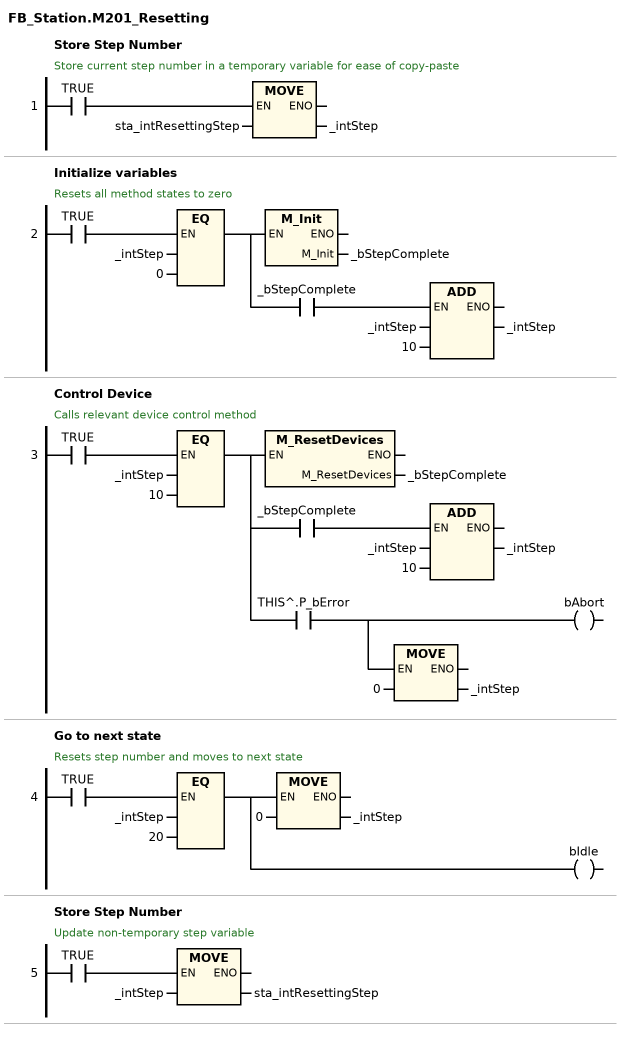
// NETWORK 1: Store Step Number
// Store current step number in a temporary variable for ease of copy-paste
_intStep := sta_intResettingStep;

// NETWORK 2: Initialize variables
// Resets all method states to zero
_w1 := _intStep = 0;
IF _w1 THEN _bStepComplete := M_Init(); END_IF
IF _w1 AND _bStepComplete THEN _intStep := _intStep + 10; END_IF

// NETWORK 3: Control Device
// Calls relevant device control method
_w2 := _intStep = 10;
IF _w2 THEN _bStepComplete := M_ResetDevices(); END_IF
IF _w2 AND _bStepComplete THEN _intStep := _intStep + 10; END_IF
_w3 := _w2 AND THIS^.P_bError;
bAbort := _w3;
IF _w3 THEN _intStep := 0; END_IF

// NETWORK 4: Go to next state
// Resets step number and moves to next state
_w4 := _intStep = 20;
IF _w4 THEN _intStep := 0; END_IF
bIdle := _w4;

// NETWORK 5: Store Step Number
// Update non-temporary step variable
sta_intResettingStep := _intStep;
END_METHOD

(* This state should make any final preparations needed for the 'Execute' state
prior to entering the 'Execute' state. *)
METHOD M301_Starting : BOOL
VAR_OUTPUT
	(* This should be set to true once the module and its components are fully
	prepared for process execution. Once set to true, the state machine will
	move to the 'Execute' state. *)
	bStarted	: BOOL;
	(* This should be set to true if an external source requests that the module
	exit its current state and come to a controlled stop. Once set to true, the
	state machine will move to the 'Stopping' state. *)
	bStop	: BOOL;
	(* This should be set to true if a potentially hazardous error or a safety
	fault has occurred in any tasks. Once set to true, the state machine will
	move to the 'Aborting' state. *)
	bAbort	: BOOL;
END_VAR
VAR
	_bStepComplete: BOOL;
	_intStep: INT;
END_VAR
VAR_INST // added by the converter: edge detectors and wires of the graphical bodies
    _w1, _w2, _w3, _w4 : BOOL;
END_VAR
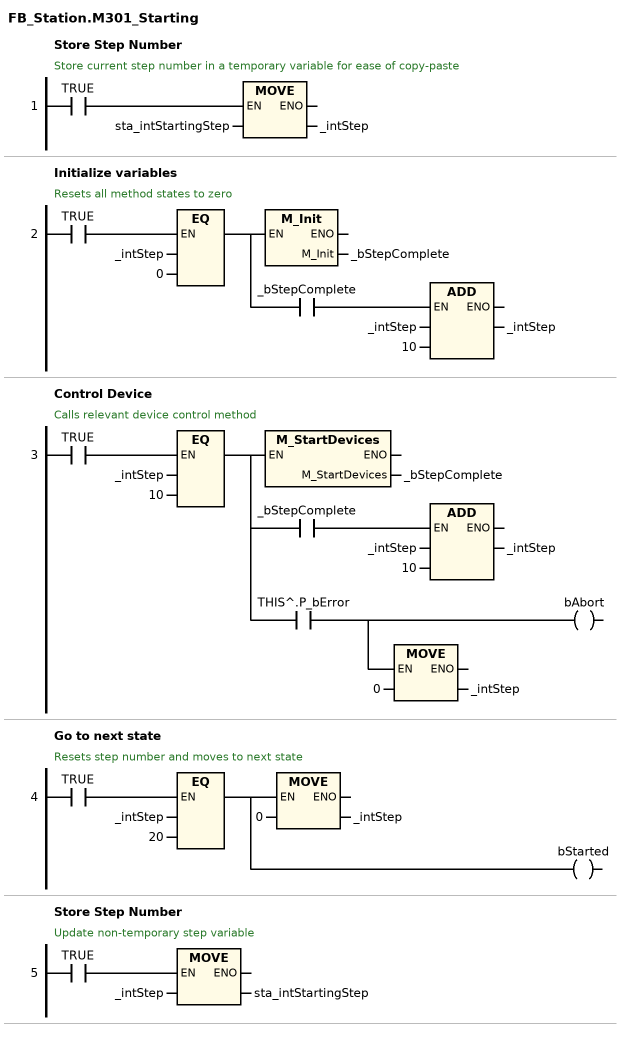
// NETWORK 1: Store Step Number
// Store current step number in a temporary variable for ease of copy-paste
_intStep := sta_intStartingStep;

// NETWORK 2: Initialize variables
// Resets all method states to zero
_w1 := _intStep = 0;
IF _w1 THEN _bStepComplete := M_Init(); END_IF
IF _w1 AND _bStepComplete THEN _intStep := _intStep + 10; END_IF

// NETWORK 3: Control Device
// Calls relevant device control method
_w2 := _intStep = 10;
IF _w2 THEN _bStepComplete := M_StartDevices(); END_IF
IF _w2 AND _bStepComplete THEN _intStep := _intStep + 10; END_IF
_w3 := _w2 AND THIS^.P_bError;
bAbort := _w3;
IF _w3 THEN _intStep := 0; END_IF

// NETWORK 4: Go to next state
// Resets step number and moves to next state
_w4 := _intStep = 20;
IF _w4 THEN _intStep := 0; END_IF
bStarted := _w4;

// NETWORK 5: Store Step Number
// Update non-temporary step variable
sta_intStartingStep := _intStep;
END_METHOD

(* This state will perform any post-execution tasks prior to moving to the
'Completed' state. *)
METHOD M321_Completing : BOOL
VAR_OUTPUT
	(* Move to the Complete state*)
	bCompleted	: BOOL;
	(* This should be set to true if an external source requests that the module
	exit its current state and come to a controlled stop. Once set to true, the
	state machine will move to the 'Stopping' state. *)
	bStop	: BOOL;
	(* This should be set to true if a potentially hazardous error or a safety
	fault has occurred in any tasks. Once set to true, the state machine will
	move to the 'Aborting' state. *)
	bAbort	: BOOL;
END_VAR
VAR
	_bStepComplete: BOOL;
	_intStep: INT;
END_VAR
VAR_INST // added by the converter: edge detectors and wires of the graphical bodies
    _w1, _w2, _w3, _w4 : BOOL;
END_VAR
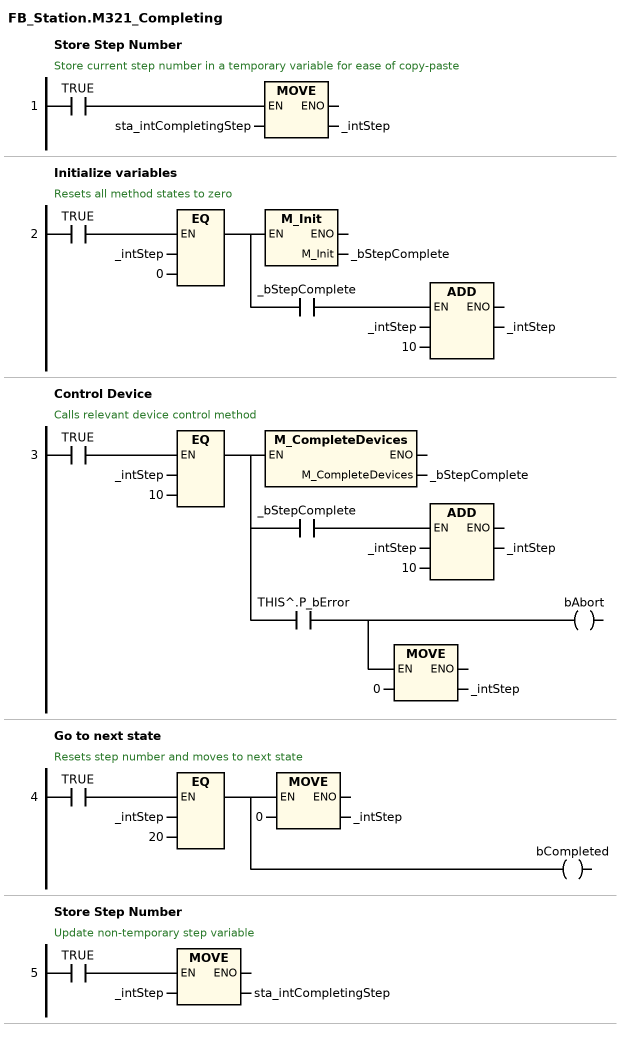
// NETWORK 1: Store Step Number
// Store current step number in a temporary variable for ease of copy-paste
_intStep := sta_intCompletingStep;

// NETWORK 2: Initialize variables
// Resets all method states to zero
_w1 := _intStep = 0;
IF _w1 THEN _bStepComplete := M_Init(); END_IF
IF _w1 AND _bStepComplete THEN _intStep := _intStep + 10; END_IF

// NETWORK 3: Control Device
// Calls relevant device control method
_w2 := _intStep = 10;
IF _w2 THEN _bStepComplete := M_CompleteDevices(); END_IF
IF _w2 AND _bStepComplete THEN _intStep := _intStep + 10; END_IF
_w3 := _w2 AND THIS^.P_bError;
bAbort := _w3;
IF _w3 THEN _intStep := 0; END_IF

// NETWORK 4: Go to next state
// Resets step number and moves to next state
_w4 := _intStep = 20;
IF _w4 THEN _intStep := 0; END_IF
bCompleted := _w4;

// NETWORK 5: Store Step Number
// Update non-temporary step variable
sta_intCompletingStep := _intStep;
END_METHOD

(* This state should safely pause task executions without completely ending or
resetting them. *)
METHOD M401_Holding : BOOL
VAR_OUTPUT
	(* This should be set to true once all execution tasks are safely paused.
	Once set to true, the state machine will move to the 'Held' state. *)
	bHeld	: BOOL;
	(* This should be set to true if an external source requests that the module
	exit its current state and come to a controlled stop. Once set to true, the
	state machine will move to the 'Stopping' state. *)
	bStop	: BOOL;
	(* This should be set to true if a potentially hazardous error or a safety
	fault has occurred in any tasks. Once set to true, the state machine will
	move to the 'Aborting' state. *)
	bAbort	: BOOL;
END_VAR
VAR
	_bStepComplete: BOOL;
	_intStep: INT;
END_VAR
VAR_INST // added by the converter: edge detectors and wires of the graphical bodies
    _w1, _w2, _w3, _w4 : BOOL;
END_VAR
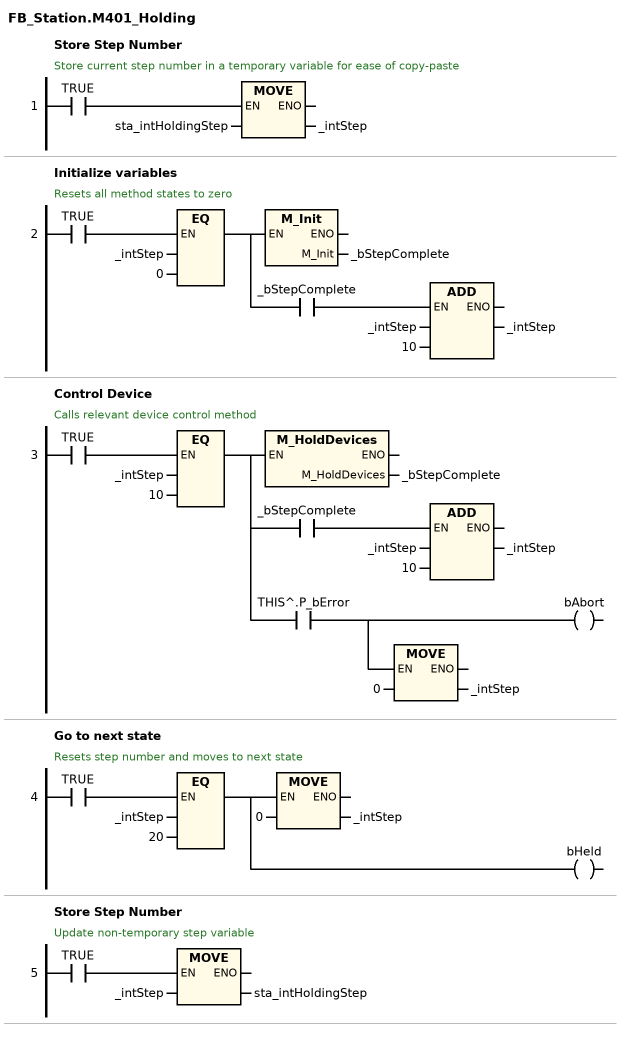
// NETWORK 1: Store Step Number
// Store current step number in a temporary variable for ease of copy-paste
_intStep := sta_intHoldingStep;

// NETWORK 2: Initialize variables
// Resets all method states to zero
_w1 := _intStep = 0;
IF _w1 THEN _bStepComplete := M_Init(); END_IF
IF _w1 AND _bStepComplete THEN _intStep := _intStep + 10; END_IF

// NETWORK 3: Control Device
// Calls relevant device control method
_w2 := _intStep = 10;
IF _w2 THEN _bStepComplete := M_HoldDevices(); END_IF
IF _w2 AND _bStepComplete THEN _intStep := _intStep + 10; END_IF
_w3 := _w2 AND THIS^.P_bError;
bAbort := _w3;
IF _w3 THEN _intStep := 0; END_IF

// NETWORK 4: Go to next state
// Resets step number and moves to next state
_w4 := _intStep = 20;
IF _w4 THEN _intStep := 0; END_IF
bHeld := _w4;

// NETWORK 5: Store Step Number
// Update non-temporary step variable
sta_intHoldingStep := _intStep;
END_METHOD

(* In this state, the module and its components should be returned to the
scenario it was in before it entered the 'Holding' step so that the
'Execute' state can pick up where it left off. *)
METHOD M421_Unholding : BOOL
VAR_OUTPUT
	(* This should be set to true once the module is ready to restart
	execution. Once set to true, the state machine will move to the 'Execute'
	state. *)
	bUnheld	: BOOL;
	(* This should be set to true if an external source requests that the module
	exit its current state and come to a controlled stop. Once set to true, the
	state machine will move to the 'Stopping' state. *)
	bStop	: BOOL;
	(* This should be set to true if a potentially hazardous error or a safety
	fault has occurred in any tasks. Once set to true, the state machine will
	move to the 'Aborting' state. *)
	bAbort	: BOOL;
END_VAR
VAR
	_bStepComplete: BOOL;
	_intStep: INT;
END_VAR
VAR_INST // added by the converter: edge detectors and wires of the graphical bodies
    _w1, _w2, _w3, _w4 : BOOL;
END_VAR
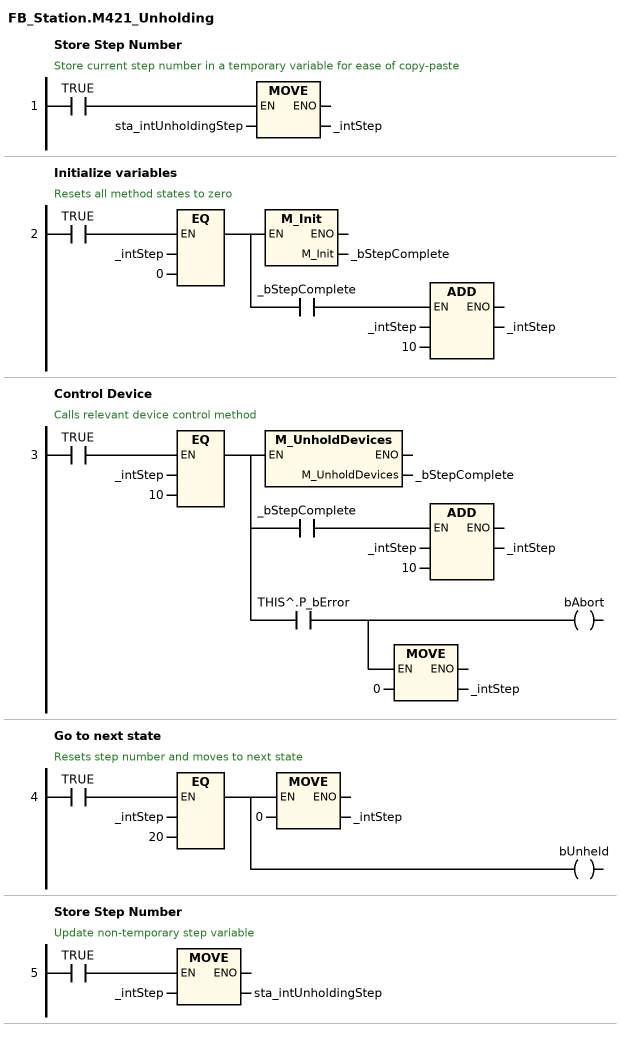
// NETWORK 1: Store Step Number
// Store current step number in a temporary variable for ease of copy-paste
_intStep := sta_intUnholdingStep;

// NETWORK 2: Initialize variables
// Resets all method states to zero
_w1 := _intStep = 0;
IF _w1 THEN _bStepComplete := M_Init(); END_IF
IF _w1 AND _bStepComplete THEN _intStep := _intStep + 10; END_IF

// NETWORK 3: Control Device
// Calls relevant device control method
_w2 := _intStep = 10;
IF _w2 THEN _bStepComplete := M_UnholdDevices(); END_IF
IF _w2 AND _bStepComplete THEN _intStep := _intStep + 10; END_IF
_w3 := _w2 AND THIS^.P_bError;
bAbort := _w3;
IF _w3 THEN _intStep := 0; END_IF

// NETWORK 4: Go to next state
// Resets step number and moves to next state
_w4 := _intStep = 20;
IF _w4 THEN _intStep := 0; END_IF
bUnheld := _w4;

// NETWORK 5: Store Step Number
// Update non-temporary step variable
sta_intUnholdingStep := _intStep;
END_METHOD

(* This state should safely pause task executions without completely ending or
resetting them. *)
METHOD M501_Suspending : BOOL
VAR_OUTPUT
	(* This should be set to true once all execution tasks are safely paused.
	Once set to true, the state machine will move to the 'Suspended' state. *)
	bSuspended	: BOOL;
	(* This should be set to true if an external source requests that the module
	exit its current state and come to a controlled stop. Once set to true, the
	state machine will move to the 'Stopping' state. *)
	bStop	: BOOL;
	(* This should be set to true if a potentially hazardous error or a safety
	fault has occurred in any tasks. Once set to true, the state machine will
	move to the 'Aborting' state. *)
	bAbort	: BOOL;
END_VAR
VAR
	_bStepComplete: BOOL;
	_intStep: INT;
END_VAR
VAR_INST // added by the converter: edge detectors and wires of the graphical bodies
    _w1, _w2, _w3, _w4 : BOOL;
END_VAR
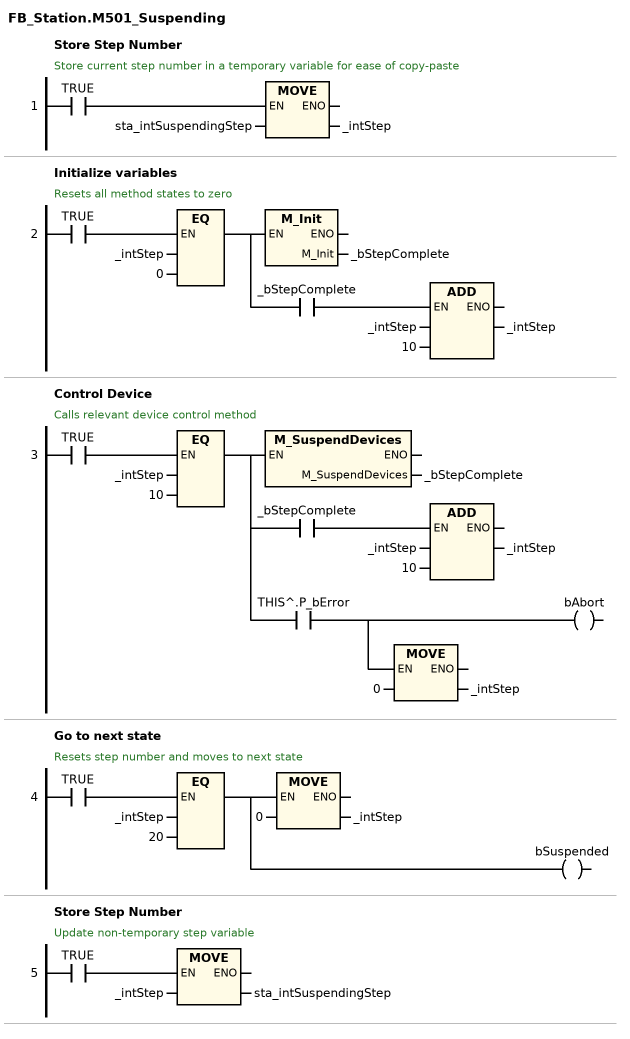
// NETWORK 1: Store Step Number
// Store current step number in a temporary variable for ease of copy-paste
_intStep := sta_intSuspendingStep;

// NETWORK 2: Initialize variables
// Resets all method states to zero
_w1 := _intStep = 0;
IF _w1 THEN _bStepComplete := M_Init(); END_IF
IF _w1 AND _bStepComplete THEN _intStep := _intStep + 10; END_IF

// NETWORK 3: Control Device
// Calls relevant device control method
_w2 := _intStep = 10;
IF _w2 THEN _bStepComplete := M_SuspendDevices(); END_IF
IF _w2 AND _bStepComplete THEN _intStep := _intStep + 10; END_IF
_w3 := _w2 AND THIS^.P_bError;
bAbort := _w3;
IF _w3 THEN _intStep := 0; END_IF

// NETWORK 4: Go to next state
// Resets step number and moves to next state
_w4 := _intStep = 20;
IF _w4 THEN _intStep := 0; END_IF
bSuspended := _w4;

// NETWORK 5: Store Step Number
// Update non-temporary step variable
sta_intSuspendingStep := _intStep;
END_METHOD

(* In this state, the module and its components should be returned to the
scenario it was in before it entered the 'Suspending' step so that the
'Execute' state can pick up where it left off. *)
METHOD M521_Unsuspending : BOOL
VAR_OUTPUT
	(* This should be set to true once the module is ready to restart
	execution. Once set to true, the state machine will move to the 'Execute'
	state. *)
	bUnsuspended	: BOOL;
	(* This should be set to true if an external source requests that the module
	exit its current state and come to a controlled stop. Once set to true, the
	state machine will move to the 'Stopping' state. *)
	bStop	: BOOL;
	(* This should be set to true if a potentially hazardous error or a safety
	fault has occurred in any tasks. Once set to true, the state machine will
	move to the 'Aborting' state. *)
	bAbort	: BOOL;
END_VAR
VAR
	_bStepComplete: BOOL;
	_intStep: INT;
END_VAR
VAR_INST // added by the converter: edge detectors and wires of the graphical bodies
    _w1, _w2, _w3, _w4 : BOOL;
END_VAR
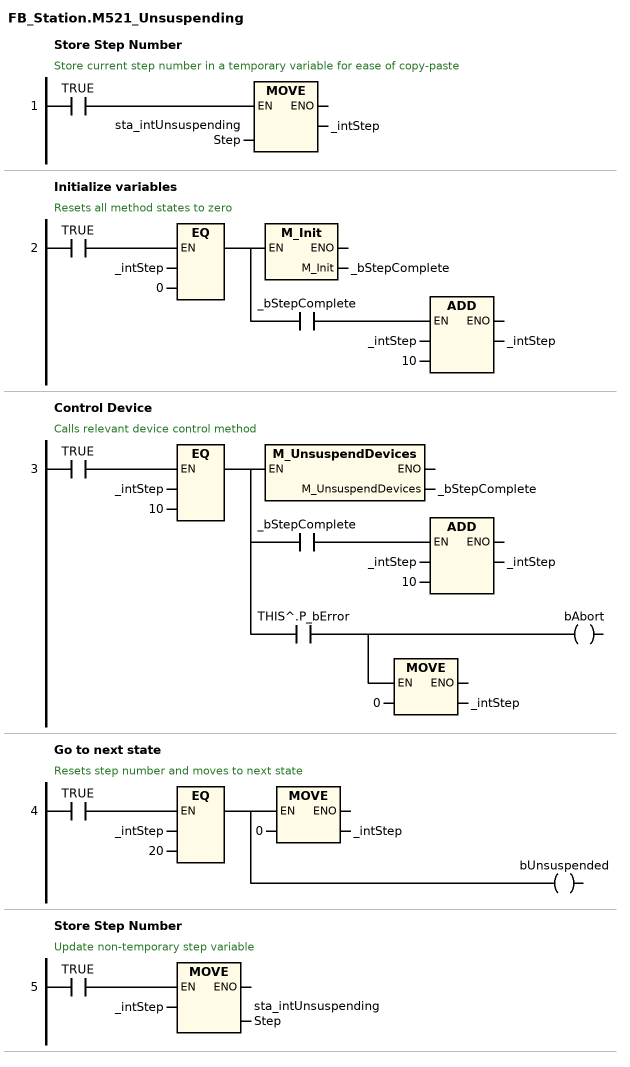
// NETWORK 1: Store Step Number
// Store current step number in a temporary variable for ease of copy-paste
_intStep := sta_intUnsuspendingStep;

// NETWORK 2: Initialize variables
// Resets all method states to zero
_w1 := _intStep = 0;
IF _w1 THEN _bStepComplete := M_Init(); END_IF
IF _w1 AND _bStepComplete THEN _intStep := _intStep + 10; END_IF

// NETWORK 3: Control Device
// Calls relevant device control method
_w2 := _intStep = 10;
IF _w2 THEN _bStepComplete := M_UnsuspendDevices(); END_IF
IF _w2 AND _bStepComplete THEN _intStep := _intStep + 10; END_IF
_w3 := _w2 AND THIS^.P_bError;
bAbort := _w3;
IF _w3 THEN _intStep := 0; END_IF

// NETWORK 4: Go to next state
// Resets step number and moves to next state
_w4 := _intStep = 20;
IF _w4 THEN _intStep := 0; END_IF
bUnsuspended := _w4;

// NETWORK 5: Store Step Number
// Update non-temporary step variable
sta_intUnsuspendingStep := _intStep;
END_METHOD

(* Calls the abort method on all devices in a station. *)
METHOD PROTECTED M_AbortDevices : BOOL
VAR CONSTANT
	_udintERROR_CODE: UDINT := E_StationError.DeviceError;
	_strERROR_MSG: T_MaxString := 'A device had an error while trying to abort!';
END_VAR
VAR_INST
	_inst_arrResults : ARRAY[1..GVL_Constants.uintMAX_STATION_DEVICE_COUNT] OF BOOL;
END_VAR
VAR
	_intStep : INT;
	_uintIndex : UINT;
	_bResult : BOOL;
	_bComplete: BOOL;
END_VAR
_bResult := FALSE;
_intStep := sta_intAbortDevicesStep;
CASE _intStep OF
	0: // Reset the results array
		FOR _uintIndex := 1 TO GVL_Constants.uintMAX_STATION_DEVICE_COUNT DO
			_inst_arrResults[_uintIndex] := FALSE;
		END_FOR
		_intStep := _intStep + 10;
	
	10: // Call the method on each device
		_bComplete := TRUE;
		FOR _uintIndex := 1 TO GVL_Constants.uintMAX_STATION_DEVICE_COUNT DO
			
			// If the method hasn't finished for this device yet, call it
			IF sta_arrDevices[_uintIndex] > 0 AND NOT _inst_arrResults[_uintIndex] THEN
				
				// Call the method
				_inst_arrResults[_uintIndex] := sta_arrDevices[_uintIndex]^.M00_Abort();
				
				// If there is an error, elevate it
				IF NOT _inst_arrResults[_uintIndex] THEN
					_bComplete := FALSE;
				END_IF
			END_IF
		END_FOR
		
		// If all methods were successful, go to the next step
		IF _bComplete THEN
			_intStep := _intStep + 10;
		END_IF
		
	20: // Return TRUE and reset
		_bResult := TRUE;
		_intStep := 0;
END_CASE
sta_intAbortDevicesStep := _intStep;
M_AbortDevices := _bResult;
END_METHOD

(* Check all devices in the device list for errors and
	raise an error if there is one. *)
METHOD PROTECTED M_CheckForDeviceErrors : BOOL
VAR_OUTPUT
	(* Unique ID of the device with an error. *)
	out_strDeviceWithError: T_MaxString;
	(* Error code on the device. *)
	out_udintErrorCode: UDINT;
	(* Error message on the device. *)
	out_strErrorMessage: T_MaxString;
END_VAR
VAR
	_uintIndex: UINT;
	_pDevice: POINTER TO FB_Device;
	_udintErrorNo: UDINT;
	_strErrorDescription: T_MaxString;
END_VAR
M_CheckForDeviceErrors := FALSE;
// Run through each device
FOR _uintIndex := 1 TO GVL_Constants.uintMAX_STATION_DEVICE_COUNT DO
	// If the pointer is set
	IF sta_arrDevices[_uintIndex] > 0 THEN
		// Get the device from the pointer
		_pDevice := sta_arrDevices[_uintIndex];
		
		// Check device for error and set error if there is one
		IF _pDevice^.P_bError THEN
			out_strDeviceWithError := _pDevice^.P_strUniqueId;
			out_udintErrorCode := _pDevice^.P_udintErrorCode;
			out_strErrorMessage := _pDevice^.P_strErrorMessage;
			M_CheckForDeviceErrors := TRUE;
			RETURN;
		END_IF
	END_IF
END_FOR
END_METHOD

(* Clears all devices set in the station. *)
METHOD PROTECTED M_ClearDevices : BOOL
VAR CONSTANT
	_udintERROR_CODE: UDINT := E_StationError.DeviceError;
	_strERROR_MSG: T_MaxString := 'A device had an error while trying to clear!';
END_VAR
VAR_INST
	_inst_arrResults : ARRAY[1..GVL_Constants.uintMAX_STATION_DEVICE_COUNT] OF BOOL;
END_VAR
VAR
	_intStep : INT;
	_uintIndex : UINT;
	_bResult : BOOL;
	_bComplete: BOOL;
END_VAR
_bResult := FALSE;
_intStep := sta_intClearDevicesStep;
CASE _intStep OF
	0: // Reset the results array
		IF NOT THIS^.P_bError THEN
			FOR _uintIndex := 1 TO GVL_Constants.uintMAX_STATION_DEVICE_COUNT DO
				_inst_arrResults[_uintIndex] := FALSE;
			END_FOR
			_intStep := _intStep + 10;
		END_IF
		
	10: // Clear module error on all devices
		FOR _uintIndex := 1 TO GVL_Constants.uintMAX_STATION_DEVICE_COUNT DO
			IF sta_arrDevices[_uintIndex] > 0 AND NOT _inst_arrResults[_uintIndex] THEN
				sta_arrDevices[_uintIndex]^.M_ClearError();
			END_IF
		END_FOR
		_intStep := _intStep + 10;
	
	20: // Call the method on each device
		_bComplete := TRUE;
		FOR _uintIndex := 1 TO GVL_Constants.uintMAX_STATION_DEVICE_COUNT DO
			
			// If the method hasn't finished for this device yet, call it
			IF sta_arrDevices[_uintIndex] > 0 AND NOT _inst_arrResults[_uintIndex] THEN
				
				// Call the method
				_inst_arrResults[_uintIndex] := sta_arrDevices[_uintIndex]^.M02_Clear();
				
				// If there is an error, elevate it
				IF sta_arrDevices[_uintIndex]^.P_bError THEN
					_bComplete := FALSE;
					THIS^.M_SetError(_udintERROR_CODE, _strERROR_MSG);
					_intStep := 0;
					
				// If the method did not complete, set complete to false
				ELSIF NOT _inst_arrResults[_uintIndex] THEN
					_bComplete := FALSE;
				END_IF
			END_IF
		END_FOR
		
		// If all methods were successful, go to the next step
		IF _bComplete THEN
			_intStep := _intStep + 10;
		END_IF
		
	30: // Return TRUE and reset
		_bResult := TRUE;
		_intStep := 0;
END_CASE
sta_intClearDevicesStep := _intStep;
M_ClearDevices := _bResult;
END_METHOD

(* Completes all devices set in the station. *)
METHOD PROTECTED M_CompleteDevices : BOOL
VAR CONSTANT
	_udintERROR_CODE: UDINT := E_StationError.DeviceError;
	_strERROR_MSG: T_MaxString := 'A device had an error while trying to complete!';
END_VAR
VAR_INST
	_inst_arrResults : ARRAY[1..GVL_Constants.uintMAX_STATION_DEVICE_COUNT] OF BOOL;
END_VAR
VAR
	_intStep : INT;
	_uintIndex : UINT;
	_bResult : BOOL;
	_bComplete: BOOL;
END_VAR
_bResult := FALSE;
_intStep := sta_intCompleteDevicesStep;
CASE _intStep OF
	0: // Reset the results array
		IF NOT THIS^.P_bError THEN
			FOR _uintIndex := 1 TO GVL_Constants.uintMAX_STATION_DEVICE_COUNT DO
				_inst_arrResults[_uintIndex] := FALSE;
			END_FOR
			_intStep := _intStep + 10;
		END_IF
	
	10: // Call the method on each device
		_bComplete := TRUE;
		FOR _uintIndex := 1 TO GVL_Constants.uintMAX_STATION_DEVICE_COUNT DO
			
			// If the method hasn't finished for this device yet, call it
			IF sta_arrDevices[_uintIndex] > 0 AND NOT _inst_arrResults[_uintIndex] THEN
				
				// Call the method
				_inst_arrResults[_uintIndex] := sta_arrDevices[_uintIndex]^.M32_Complete();
				
				// If there is an error, elevate it
				IF sta_arrDevices[_uintIndex]^.P_bError THEN
					_bComplete := FALSE;
					THIS^.M_SetError(_udintERROR_CODE, _strERROR_MSG);
					_intStep := 0;
					
				// If the method did not complete, set complete to false
				ELSIF NOT _inst_arrResults[_uintIndex] THEN
					_bComplete := FALSE;
				END_IF
			END_IF
		END_FOR
		
		// If all methods were successful, go to the next step
		IF _bComplete THEN
			_intStep := _intStep + 10;
		END_IF
		
	20: // Return TRUE and reset
		_bResult := TRUE;
		_intStep := 0;
END_CASE
sta_intCompleteDevicesStep := _intStep;
M_CompleteDevices := _bResult;
END_METHOD

(* Holds all devices set in the station. *)
METHOD PROTECTED M_HoldDevices : BOOL
VAR CONSTANT
	_udintERROR_CODE: UDINT := E_StationError.DeviceError;
	_strERROR_MSG: T_MaxString := 'A device had an error while trying to hold!';
END_VAR
VAR_INST
	_inst_arrResults : ARRAY[1..GVL_Constants.uintMAX_STATION_DEVICE_COUNT] OF BOOL;
END_VAR
VAR
	_intStep : INT;
	_uintIndex : UINT;
	_bResult : BOOL;
	_bComplete: BOOL;
END_VAR
_bResult := FALSE;
_intStep := sta_intHoldDevicesStep;
CASE _intStep OF
	0: // Reset the results array
		IF NOT THIS^.P_bError THEN
			FOR _uintIndex := 1 TO GVL_Constants.uintMAX_STATION_DEVICE_COUNT DO
				_inst_arrResults[_uintIndex] := FALSE;
			END_FOR
			_intStep := _intStep + 10;
		END_IF
	
	10: // Call the method on each device
		_bComplete := TRUE;
		FOR _uintIndex := 1 TO GVL_Constants.uintMAX_STATION_DEVICE_COUNT DO
			
			// If the method hasn't finished for this device yet, call it
			IF sta_arrDevices[_uintIndex] > 0 AND NOT _inst_arrResults[_uintIndex] THEN
				
				// Call the method
				_inst_arrResults[_uintIndex] := sta_arrDevices[_uintIndex]^.M40_Hold();
				
				// If there is an error, elevate it
				IF sta_arrDevices[_uintIndex]^.P_bError THEN
					_bComplete := FALSE;
					THIS^.M_SetError(_udintERROR_CODE, _strERROR_MSG);
					_intStep := 0;
					
				// If the method did not complete, set complete to false
				ELSIF NOT _inst_arrResults[_uintIndex] THEN
					_bComplete := FALSE;
				END_IF
			END_IF
		END_FOR
		
		// If all methods were successful, go to the next step
		IF _bComplete THEN
			_intStep := _intStep + 10;
		END_IF
		
	20: // Return TRUE and reset
		_bResult := TRUE;
		_intStep := 0;
END_CASE
sta_intHoldDevicesStep := _intStep;
M_HoldDevices := _bResult;
END_METHOD

(* Resets all devices set in the station. *)
METHOD PROTECTED M_ResetDevices : BOOL
VAR CONSTANT
	_udintERROR_CODE: UDINT := E_StationError.DeviceError;
	_strERROR_MSG: T_MaxString := 'A device had an error while trying to reset!';
END_VAR
VAR_INST
	_inst_arrResults : ARRAY[1..GVL_Constants.uintMAX_STATION_DEVICE_COUNT] OF BOOL;
END_VAR
VAR
	_intStep : INT;
	_uintIndex : UINT;
	_bResult : BOOL;
	_bComplete: BOOL;
END_VAR
_bResult := FALSE;
_intStep := sta_intResetDevicesStep;
CASE _intStep OF
	0: // Reset the results array
		IF NOT THIS^.P_bError THEN
			FOR _uintIndex := 1 TO GVL_Constants.uintMAX_STATION_DEVICE_COUNT DO
				_inst_arrResults[_uintIndex] := FALSE;
			END_FOR
			_intStep := _intStep + 10;
		END_IF
	
	10: // Call the method on each device
		_bComplete := TRUE;
		FOR _uintIndex := 1 TO GVL_Constants.uintMAX_STATION_DEVICE_COUNT DO
			
			// If the method hasn't finished for this device yet, call it
			IF sta_arrDevices[_uintIndex] > 0 AND NOT _inst_arrResults[_uintIndex] THEN
				
				// Call the method
				_inst_arrResults[_uintIndex] := sta_arrDevices[_uintIndex]^.M20_Reset();
				
				// If there is an error, elevate it
				IF sta_arrDevices[_uintIndex]^.P_bError THEN
					_bComplete := FALSE;
					THIS^.M_SetError(_udintERROR_CODE, _strERROR_MSG);
					_intStep := 0;
					
				// If the method did not complete, set complete to false
				ELSIF NOT _inst_arrResults[_uintIndex] THEN
					_bComplete := FALSE;
				END_IF
			END_IF
		END_FOR
		
		// If all methods were successful, go to the next step
		IF _bComplete THEN
			_intStep := _intStep + 10;
		END_IF
		
	20: // Return TRUE and reset
		_bResult := TRUE;
		_intStep := 0;
END_CASE
sta_intResetDevicesStep := _intStep;
M_ResetDevices := _bResult;
END_METHOD

(* Starts all devices set in the station. *)
METHOD PROTECTED M_StartDevices : BOOL
VAR CONSTANT
	_udintERROR_CODE: UDINT := E_StationError.DeviceError;
	_strERROR_MSG: T_MaxString := 'A device had an error while trying to start!';
END_VAR
VAR_INST
	_inst_arrResults : ARRAY[1..GVL_Constants.uintMAX_STATION_DEVICE_COUNT] OF BOOL;
END_VAR
VAR
	_intStep : INT;
	_uintIndex : UINT;
	_bResult : BOOL;
	_bComplete: BOOL;
END_VAR
_bResult := FALSE;
_intStep := sta_intStartDevicesStep;
CASE _intStep OF
	0: // Reset the results array
		IF NOT THIS^.P_bError THEN
			FOR _uintIndex := 1 TO GVL_Constants.uintMAX_STATION_DEVICE_COUNT DO
				_inst_arrResults[_uintIndex] := FALSE;
			END_FOR
			_intStep := _intStep + 10;
		END_IF
	
	10: // Call the method on each device
		_bComplete := TRUE;
		FOR _uintIndex := 1 TO GVL_Constants.uintMAX_STATION_DEVICE_COUNT DO
			
			// If the method hasn't finished for this device yet, call it
			IF sta_arrDevices[_uintIndex] > 0 AND NOT _inst_arrResults[_uintIndex] THEN
				
				// Call the method
				_inst_arrResults[_uintIndex] := sta_arrDevices[_uintIndex]^.M30_Start();
				
				// If there is an error, elevate it
				IF sta_arrDevices[_uintIndex]^.P_bError THEN
					_bComplete := FALSE;
					THIS^.M_SetError(_udintERROR_CODE, _strERROR_MSG);
					_intStep := 0;
					
				// If the method did not complete, set complete to false
				ELSIF NOT _inst_arrResults[_uintIndex] THEN
					_bComplete := FALSE;
				END_IF
			END_IF
		END_FOR
		
		// If all methods were successful, go to the next step
		IF _bComplete THEN
			_intStep := _intStep + 10;
		END_IF
		
	20: // Return TRUE and reset
		_bResult := TRUE;
		_intStep := 0;
END_CASE
sta_intStartDevicesStep := _intStep;
M_StartDevices := _bResult;
END_METHOD

(* Stops all devices set in the station. *)
METHOD PROTECTED M_StopDevices : BOOL
VAR CONSTANT
	_udintERROR_CODE: UDINT := E_StationError.DeviceError;
	_strERROR_MSG: T_MaxString := 'A device had an error while trying to stop!';
END_VAR
VAR_INST
	_inst_arrResults : ARRAY[1..GVL_Constants.uintMAX_STATION_DEVICE_COUNT] OF BOOL;
END_VAR
VAR
	_intStep : INT;
	_uintIndex : UINT;
	_bResult : BOOL;
	_bComplete: BOOL;
END_VAR
_bResult := FALSE;
_intStep := sta_intStopDevicesStep;
CASE _intStep OF
	0: // Reset the results array
		IF NOT THIS^.P_bError THEN
			FOR _uintIndex := 1 TO GVL_Constants.uintMAX_STATION_DEVICE_COUNT DO
				_inst_arrResults[_uintIndex] := FALSE;
			END_FOR
			_intStep := _intStep + 10;
		END_IF
	
	10: // Call the method on each device
		_bComplete := TRUE;
		FOR _uintIndex := 1 TO GVL_Constants.uintMAX_STATION_DEVICE_COUNT DO
			
			// If the method hasn't finished for this device yet, call it
			IF sta_arrDevices[_uintIndex] > 0 AND NOT _inst_arrResults[_uintIndex] THEN
				
				// Call the method
				_inst_arrResults[_uintIndex] := sta_arrDevices[_uintIndex]^.M10_Stop();
				
				// If there is an error, elevate it
				IF sta_arrDevices[_uintIndex]^.P_bError THEN
					_bComplete := FALSE;
					THIS^.M_SetError(_udintERROR_CODE, _strERROR_MSG);
					_intStep := 0;
					
				// If the method did not complete, set complete to false
				ELSIF NOT _inst_arrResults[_uintIndex] THEN
					_bComplete := FALSE;
				END_IF
			END_IF
		END_FOR
		
		// If all methods were successful, go to the next step
		IF _bComplete THEN
			_intStep := _intStep + 10;
		END_IF
		
	20: // Return TRUE and reset
		_bResult := TRUE;
		_intStep := 0;
END_CASE
sta_intStopDevicesStep := _intStep;
M_StopDevices := _bResult;
END_METHOD

(* Suspends all devices set in the station. *)
METHOD PROTECTED M_SuspendDevices : BOOL
VAR CONSTANT
	_udintERROR_CODE: UDINT := E_StationError.DeviceError;
	_strERROR_MSG: T_MaxString := 'A device had an error while trying to suspend!';
END_VAR
VAR_INST
	_inst_arrResults : ARRAY[1..GVL_Constants.uintMAX_STATION_DEVICE_COUNT] OF BOOL;
END_VAR
VAR
	_intStep : INT;
	_uintIndex : UINT;
	_bResult : BOOL;
	_bComplete: BOOL;
END_VAR
_bResult := FALSE;
_intStep := sta_intSuspendDevicesStep;
CASE _intStep OF
	0: // Reset the results array
		IF NOT THIS^.P_bError THEN
			FOR _uintIndex := 1 TO GVL_Constants.uintMAX_STATION_DEVICE_COUNT DO
				_inst_arrResults[_uintIndex] := FALSE;
			END_FOR
			_intStep := _intStep + 10;
		END_IF
	
	10: // Call the method on each device
		_bComplete := TRUE;
		FOR _uintIndex := 1 TO GVL_Constants.uintMAX_STATION_DEVICE_COUNT DO
			
			// If the method hasn't finished for this device yet, call it
			IF sta_arrDevices[_uintIndex] > 0 AND NOT _inst_arrResults[_uintIndex] THEN
				
				// Call the method
				_inst_arrResults[_uintIndex] := sta_arrDevices[_uintIndex]^.M50_Suspend();
				
				// If there is an error, elevate it
				IF sta_arrDevices[_uintIndex]^.P_bError THEN
					_bComplete := FALSE;
					THIS^.M_SetError(_udintERROR_CODE, _strERROR_MSG);
					_intStep := 0;
					
				// If the method did not complete, set complete to false
				ELSIF NOT _inst_arrResults[_uintIndex] THEN
					_bComplete := FALSE;
				END_IF
			END_IF
		END_FOR
		
		// If all methods were successful, go to the next step
		IF _bComplete THEN
			_intStep := _intStep + 10;
		END_IF
		
	20: // Return TRUE and reset
		_bResult := TRUE;
		_intStep := 0;
END_CASE
sta_intSuspendDevicesStep := _intStep;
M_SuspendDevices := _bResult;
END_METHOD

(* Unholds all devices set in the station. *)
METHOD PROTECTED M_UnholdDevices : BOOL
VAR CONSTANT
	_udintERROR_CODE: UDINT := E_StationError.DeviceError;
	_strERROR_MSG: T_MaxString := 'A device had an error while trying to unhold!';
END_VAR
VAR_INST
	_inst_arrResults : ARRAY[1..GVL_Constants.uintMAX_STATION_DEVICE_COUNT] OF BOOL;
END_VAR
VAR
	_intStep : INT;
	_uintIndex : UINT;
	_bResult : BOOL;
	_bComplete: BOOL;
END_VAR
_bResult := FALSE;
_intStep := sta_intUnholdDevicesStep;
CASE _intStep OF
	0: // Reset the results array
		IF NOT THIS^.P_bError THEN
			FOR _uintIndex := 1 TO GVL_Constants.uintMAX_STATION_DEVICE_COUNT DO
				_inst_arrResults[_uintIndex] := FALSE;
			END_FOR
			_intStep := _intStep + 10;
		END_IF
	
	10: // Call the method on each device
		_bComplete := TRUE;
		FOR _uintIndex := 1 TO GVL_Constants.uintMAX_STATION_DEVICE_COUNT DO
			
			// If the method hasn't finished for this device yet, call it
			IF sta_arrDevices[_uintIndex] > 0 AND NOT _inst_arrResults[_uintIndex] THEN
				
				// Call the method
				_inst_arrResults[_uintIndex] := sta_arrDevices[_uintIndex]^.M42_Unhold();
				
				// If there is an error, elevate it
				IF sta_arrDevices[_uintIndex]^.P_bError THEN
					_bComplete := FALSE;
					THIS^.M_SetError(_udintERROR_CODE, _strERROR_MSG);
					_intStep := 0;
					
				// If the method did not complete, set complete to false
				ELSIF NOT _inst_arrResults[_uintIndex] THEN
					_bComplete := FALSE;
				END_IF
			END_IF
		END_FOR
		
		// If all methods were successful, go to the next step
		IF _bComplete THEN
			_intStep := _intStep + 10;
		END_IF
		
	20: // Return TRUE and reset
		_bResult := TRUE;
		_intStep := 0;
END_CASE
sta_intUnholdDevicesStep := _intStep;
M_UnholdDevices := _bResult;
END_METHOD

(* Unsuspends all devices set in the station. *)
METHOD PROTECTED M_UnsuspendDevices : BOOL
VAR CONSTANT
	_udintERROR_CODE: UDINT := E_StationError.DeviceError;
	_strERROR_MSG: T_MaxString := 'A device had an error while trying to unsuspend!';
END_VAR
VAR_INST
	_inst_arrResults : ARRAY[1..GVL_Constants.uintMAX_STATION_DEVICE_COUNT] OF BOOL;
END_VAR
VAR
	_intStep : INT;
	_uintIndex : UINT;
	_bResult : BOOL;
	_bComplete: BOOL;
END_VAR
_bResult := FALSE;
_intStep := sta_intUnsuspendDevicesStep;
CASE _intStep OF
	0: // Reset the results array
		IF NOT THIS^.P_bError THEN
			FOR _uintIndex := 1 TO GVL_Constants.uintMAX_STATION_DEVICE_COUNT DO
				_inst_arrResults[_uintIndex] := FALSE;
			END_FOR
			_intStep := _intStep + 10;
		END_IF
	
	10: // Call the method on each device
		_bComplete := TRUE;
		FOR _uintIndex := 1 TO GVL_Constants.uintMAX_STATION_DEVICE_COUNT DO
			
			// If the method hasn't finished for this device yet, call it
			IF sta_arrDevices[_uintIndex] > 0 AND NOT _inst_arrResults[_uintIndex] THEN
				
				// Call the method
				_inst_arrResults[_uintIndex] := sta_arrDevices[_uintIndex]^.M52_Unsuspend();
				
				// If there is an error, elevate it
				IF sta_arrDevices[_uintIndex]^.P_bError THEN
					_bComplete := FALSE;
					THIS^.M_SetError(_udintERROR_CODE, _strERROR_MSG);
					_intStep := 0;
					
				// If the method did not complete, set complete to false
				ELSIF NOT _inst_arrResults[_uintIndex] THEN
					_bComplete := FALSE;
				END_IF
			END_IF
		END_FOR
		
		// If all methods were successful, go to the next step
		IF _bComplete THEN
			_intStep := _intStep + 10;
		END_IF
		
	20: // Return TRUE and reset
		_bResult := TRUE;
		_intStep := 0;
END_CASE
sta_intUnsuspendDevicesStep := _intStep;
M_UnsuspendDevices := _bResult;
END_METHOD

(* Sets a device in the device list. *)
METHOD PROTECTED M_SetDevice : BOOL
VAR_INPUT
	(* Index of device to set. Between 1 and uintMAX_STATION_DEVICE_COUNT. *)
	_in_uintIndex : UINT;
	(* Reference to the device to add to the device array. *)
	_in_fbDevice : REFERENCE TO FB_Device;
END_VAR

VAR
	_pController: POINTER TO FB_DeviceController;
END_VAR
M_SetDevice := FALSE;
// Check that the index is valid
IF _in_uintIndex > 0 AND _in_uintIndex <= GVL_Constants.uintMAX_STATION_DEVICE_COUNT THEN
	
	// Check that the reference is valid
	IF __ISVALIDREF(_in_fbDevice) THEN
		
		// Get the controller if created
		IF sta_arrDevices[_in_uintIndex] > 0 THEN
			_pController := sta_arrDevices[_in_uintIndex];
			
		// Else create it
		ELSE
			_pController := __NEW(FB_DeviceController);
			THIS^.M_LogMessage(CONCAT('Created controller for ', _in_fbDevice.P_strUniqueId));
		END_IF
		
		// Call the controller
		_pController^(
			in_strUniqueId := CONCAT(_in_fbDevice.P_strUniqueId, '::Controller'),
			in_pDevice := ADR(_in_fbDevice));
		sta_arrDevices[_in_uintIndex] := _pController;
		M_SetDevice := TRUE;
	END_IF
END_IF
END_METHOD

(* The array of device pointers for this station. *)
PROPERTY P_arrDevices : T_StationDeviceArray
GET
P_arrDevices := sta_arrDevices;
END_GET
END_PROPERTY

(* Resets all state step numbers. *)
METHOD PRIVATE M_Init : BOOL
VAR_INPUT
END_VAR
sta_intAbortDevicesStep:=0;
sta_intClearDevicesStep:=0;
sta_intCompleteDevicesStep:=0;
sta_intHoldDevicesStep:=0;
sta_intResetDevicesStep:=0;
sta_intStartDevicesStep:=0;
sta_intStopDevicesStep:=0;
sta_intSuspendDevicesStep:=0;
sta_intUnholdDevicesStep:=0;
sta_intUnsuspendDevicesStep:=0;

sta_intAbortingStep:=0;
sta_intClearingStep:=0;
sta_intResettingStep:=0;
sta_intStartingStep:=0;
sta_intCompletingStep:=0;
sta_intHoldingStep:=0;
sta_intUnholdingStep:=0;
sta_intSuspendingStep:=0;
sta_intUnsuspendingStep:=0;
sta_intStoppingStep:=0;

M_Init := TRUE;
END_METHOD

METHOD FB_exit : BOOL
VAR_INPUT
	bInCopyCode : BOOL; 
END_VAR

VAR
	_uintIndex: UINT;
END_VAR
FOR _uintIndex := 1 TO GVL_Constants.uintMAX_STATION_DEVICE_COUNT DO
	IF sta_arrDevices[_uintIndex] > 0 THEN
		__DELETE(sta_arrDevices[_uintIndex]);
	END_IF
END_FOR
END_METHOD

END_FUNCTION_BLOCK

// Concrete/FB_DeviceController
(* Controller implementing the standard process for using the
	generic device interfaces within a station. *)
{attribute 'enable_dynamic_creation'}
FUNCTION_BLOCK FB_DeviceController EXTENDS FB_Module
VAR_INPUT
	(* Pointer to the device to control. *)
	in_pDevice : POINTER TO FB_Device;
END_VAR
VAR_OUTPUT
END_VAR
VAR
	intAbortStep: INT;
	intClearStep: INT;
	intCompleteStep: INT;
	intHoldStep: INT;
	intResetStep: INT;
	intStartStep: INT;
	intStopStep: INT;
	intSuspendStep: INT;
	intUnholdStep: INT;
	intUnsuspendStep: INT;
END_VAR

// Reinitializes all variables
METHOD PRIVATE M_Init : BOOL
VAR_INPUT
END_VAR
VAR
END_VAR
intAbortStep := 0;
intClearStep := 0;
intCompleteStep := 0;
intHoldStep := 0;
intResetStep := 0;
intStartStep := 0;
intStopStep := 0;
intSuspendStep := 0;
intUnholdStep := 0;
intUnsuspendStep := 0;
M_Init := TRUE;
END_METHOD

(* Aborts the device then returns TRUE once aborted. *)
METHOD M00_Abort : BOOL
VAR CONSTANT
	_intFINAL_STEP : INT := 1000;
	_strSTART_MSG: T_MaxString := 'Aborting device';
	_strFINISH_MSG: T_MaxString := 'Device aborted';
END_VAR
VAR
	_bStepComplete: BOOL;
	_intStep: INT;
END_VAR
VAR_INST // added by the converter: edge detectors and wires of the graphical bodies
    _w1, _w2, _w3, _w4, _w5, _w6 : BOOL;
END_VAR
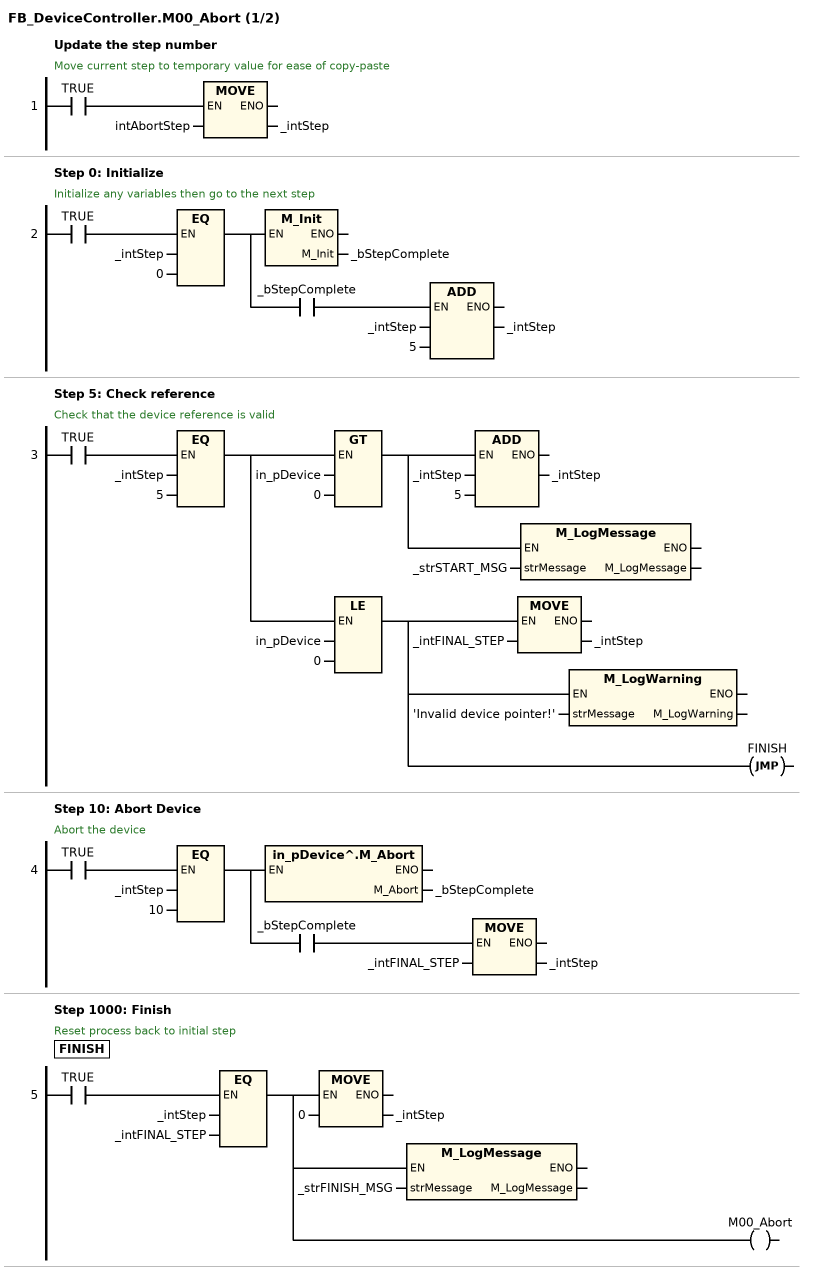
// NETWORK 1: Update the step number
// Move current step to temporary value for ease of copy-paste
_intStep := intAbortStep;

// NETWORK 2: Step 0: Initialize
// Initialize any variables then go to the next step
_w1 := _intStep = 0;
IF _w1 THEN _bStepComplete := M_Init(); END_IF
IF _w1 AND _bStepComplete THEN _intStep := _intStep + 5; END_IF

// NETWORK 3: Step 5: Check reference
// Check that the device reference is valid
_w2 := _intStep = 5;
_w3 := _w2 AND in_pDevice > 0;
IF _w3 THEN _intStep := _intStep + 5; END_IF
IF _w3 THEN M_LogMessage(strMessage := _strSTART_MSG); END_IF
_w4 := _w2 AND in_pDevice <= 0;
IF _w4 THEN _intStep := _intFINAL_STEP; END_IF
IF _w4 THEN M_LogWarning(strMessage := 'Invalid device pointer!'); END_IF
IF _w4 THEN JMP FINISH; END_IF

// NETWORK 4: Step 10: Abort Device
// Abort the device
_w5 := _intStep = 10;
IF _w5 THEN _bStepComplete := in_pDevice^.M_Abort(); END_IF
IF _w5 AND _bStepComplete THEN _intStep := _intFINAL_STEP; END_IF

// NETWORK 5: Step 1000: Finish
// Reset process back to initial step
FINISH:
_w6 := _intStep = _intFINAL_STEP;
IF _w6 THEN _intStep := 0; END_IF
IF _w6 THEN M_LogMessage(strMessage := _strFINISH_MSG); END_IF
M00_Abort := _w6;

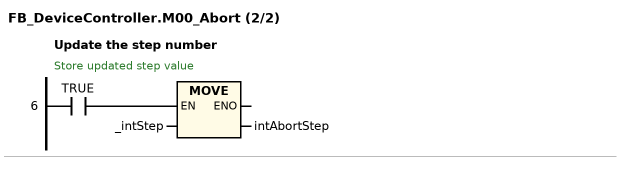
// NETWORK 6: Update the step number
// Store updated step value
intAbortStep := _intStep;
END_METHOD

(* Clears errors on the device then returns TRUE once cleared. *)
METHOD M02_Clear : BOOL
VAR CONSTANT
	_intFINAL_STEP : INT := 1000;
	_intERROR_STEP : INT := 2000;
	_udintERROR_CODE: UDINT := E_DeviceControllerError.ClearError;
	_strERROR_MSG: T_MaxString := 'Error while trying to clear device!';
	_strSTART_MSG: T_MaxString := 'Clearing device';
	_strFINISH_MSG: T_MaxString := 'Device cleared';
END_VAR
VAR
	_bStepComplete: BOOL;
	_intStep: INT;
END_VAR
VAR_INST // added by the converter: edge detectors and wires of the graphical bodies
    _w1, _w2, _w3, _w4, _w5, _w6, _w7, _w8 : BOOL;
END_VAR
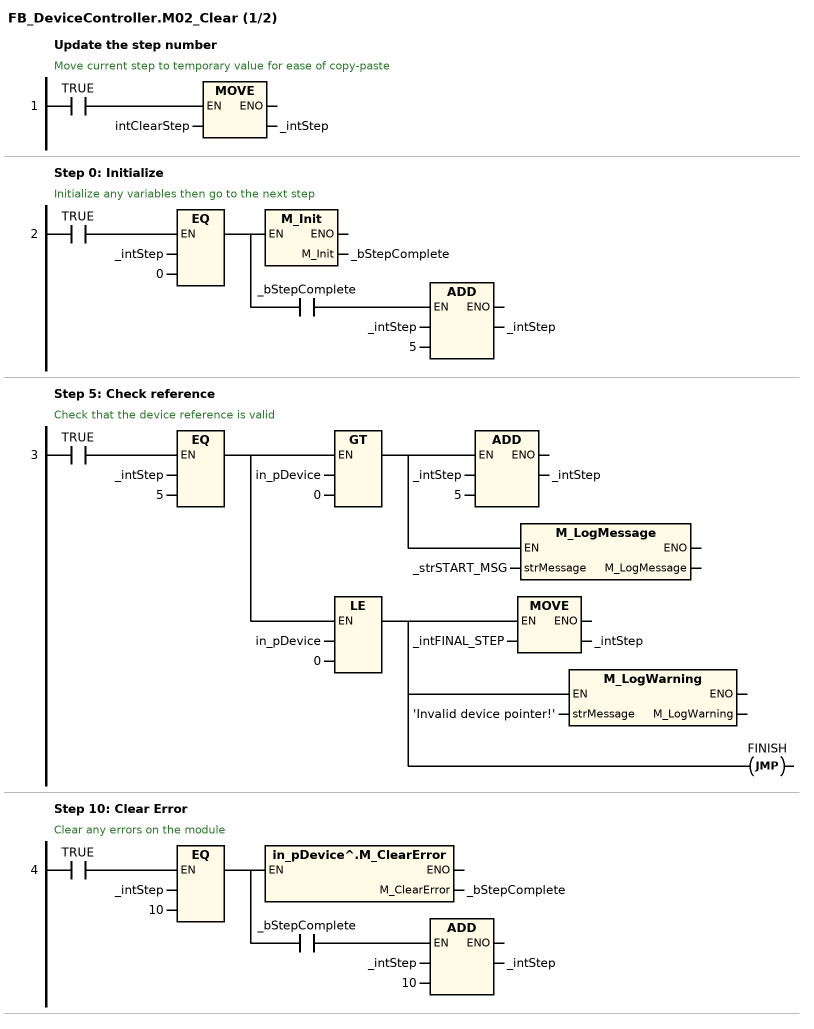
// NETWORK 1: Update the step number
// Move current step to temporary value for ease of copy-paste
_intStep := intClearStep;

// NETWORK 2: Step 0: Initialize
// Initialize any variables then go to the next step
_w1 := _intStep = 0;
IF _w1 THEN _bStepComplete := M_Init(); END_IF
IF _w1 AND _bStepComplete THEN _intStep := _intStep + 5; END_IF

// NETWORK 3: Step 5: Check reference
// Check that the device reference is valid
_w2 := _intStep = 5;
_w3 := _w2 AND in_pDevice > 0;
IF _w3 THEN _intStep := _intStep + 5; END_IF
IF _w3 THEN M_LogMessage(strMessage := _strSTART_MSG); END_IF
_w4 := _w2 AND in_pDevice <= 0;
IF _w4 THEN _intStep := _intFINAL_STEP; END_IF
IF _w4 THEN M_LogWarning(strMessage := 'Invalid device pointer!'); END_IF
IF _w4 THEN JMP FINISH; END_IF

// NETWORK 4: Step 10: Clear Error
// Clear any errors on the module
_w5 := _intStep = 10;
IF _w5 THEN _bStepComplete := in_pDevice^.M_ClearError(); END_IF
IF _w5 AND _bStepComplete THEN _intStep := _intStep + 10; END_IF

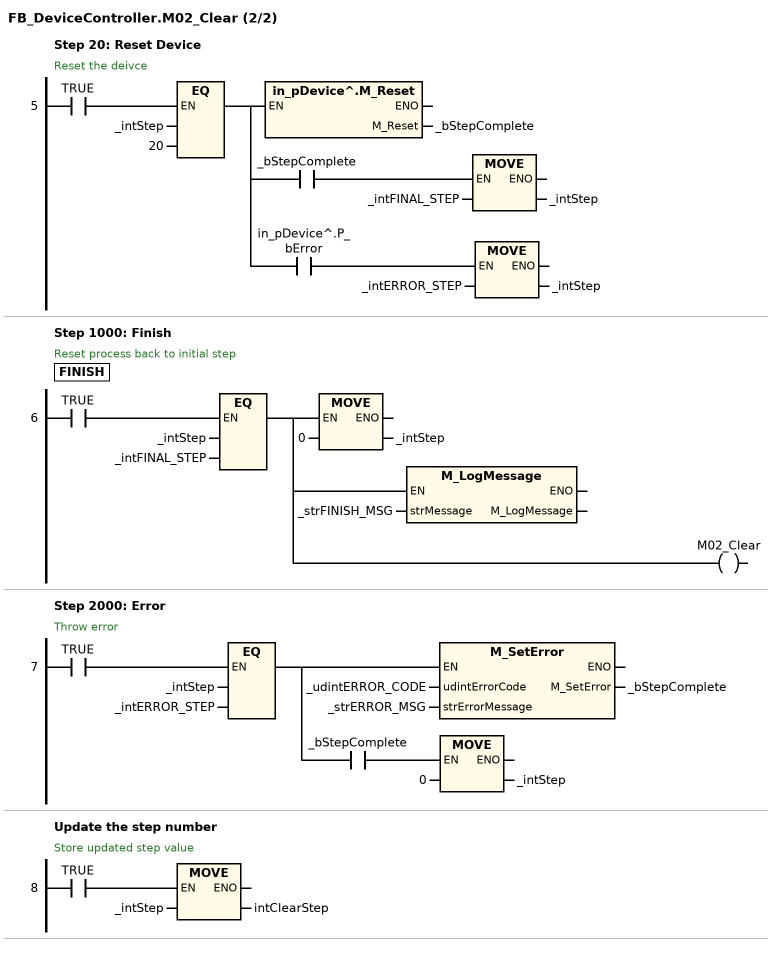
// NETWORK 5: Step 20: Reset Device
// Reset the deivce
_w6 := _intStep = 20;
IF _w6 THEN _bStepComplete := in_pDevice^.M_Reset(); END_IF
IF _w6 AND _bStepComplete THEN _intStep := _intFINAL_STEP; END_IF
IF _w6 AND in_pDevice^.P_bError THEN _intStep := _intERROR_STEP; END_IF

// NETWORK 6: Step 1000: Finish
// Reset process back to initial step
FINISH:
_w7 := _intStep = _intFINAL_STEP;
IF _w7 THEN _intStep := 0; END_IF
IF _w7 THEN M_LogMessage(strMessage := _strFINISH_MSG); END_IF
M02_Clear := _w7;

// NETWORK 7: Step 2000: Error
// Throw error
_w8 := _intStep = _intERROR_STEP;
IF _w8 THEN
    _bStepComplete := M_SetError(udintErrorCode := _udintERROR_CODE, strErrorMessage := _strERROR_MSG);
END_IF
IF _w8 AND _bStepComplete THEN _intStep := 0; END_IF

// NETWORK 8: Update the step number
// Store updated step value
intClearStep := _intStep;
END_METHOD

(* Stops the device then returns TRUE. *)
METHOD M10_Stop : BOOL
VAR CONSTANT
	_intFINAL_STEP : INT := 1000;
	_intERROR_STEP : INT := 2000;
	_udintERROR_CODE: UDINT := E_DeviceControllerError.StopError;
	_strERROR_MSG: T_MaxString := 'Error while trying to stop device!';
	_strSTART_MSG: T_MaxString := 'Stopping device';
	_strFINISH_MSG: T_MaxString := 'Device stopped';
END_VAR
VAR
	_bStepComplete: BOOL;
	_intStep: INT;
	_bConnected: BOOL;
END_VAR
VAR_INST // added by the converter: edge detectors and wires of the graphical bodies
    _w1, _w2, _w3, _w4, _w5, _w6, _w7, _w8, _w9, _w10, _w11, _w12 : BOOL;
END_VAR
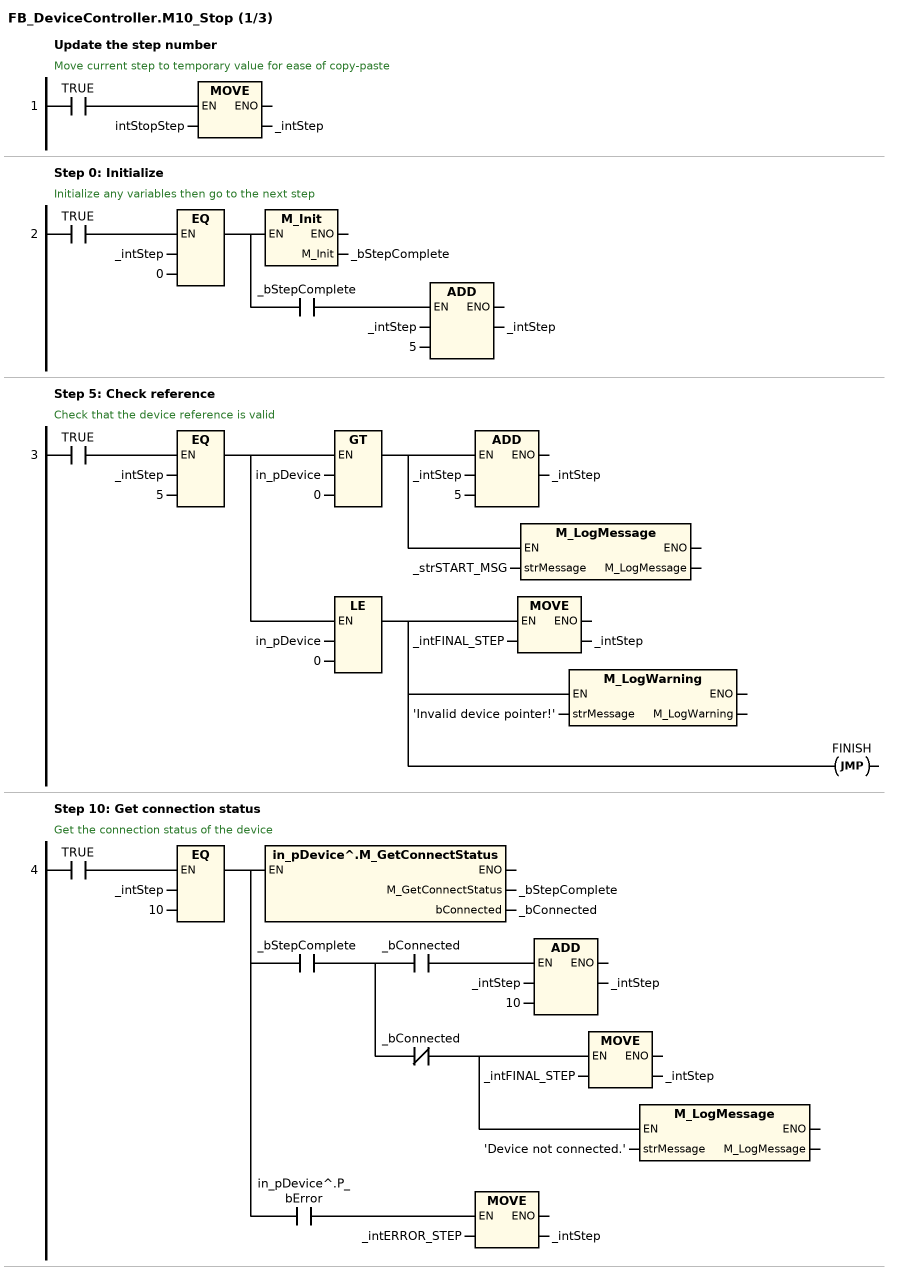
// NETWORK 1: Update the step number
// Move current step to temporary value for ease of copy-paste
_intStep := intStopStep;

// NETWORK 2: Step 0: Initialize
// Initialize any variables then go to the next step
_w1 := _intStep = 0;
IF _w1 THEN _bStepComplete := M_Init(); END_IF
IF _w1 AND _bStepComplete THEN _intStep := _intStep + 5; END_IF

// NETWORK 3: Step 5: Check reference
// Check that the device reference is valid
_w2 := _intStep = 5;
_w3 := _w2 AND in_pDevice > 0;
IF _w3 THEN _intStep := _intStep + 5; END_IF
IF _w3 THEN M_LogMessage(strMessage := _strSTART_MSG); END_IF
_w4 := _w2 AND in_pDevice <= 0;
IF _w4 THEN _intStep := _intFINAL_STEP; END_IF
IF _w4 THEN M_LogWarning(strMessage := 'Invalid device pointer!'); END_IF
IF _w4 THEN JMP FINISH; END_IF

// NETWORK 4: Step 10: Get connection status
// Get the connection status of the device
_w5 := _intStep = 10;
IF _w5 THEN _bStepComplete := in_pDevice^.M_GetConnectStatus(bConnected => _bConnected); END_IF
_w6 := _w5 AND _bStepComplete;
IF _w6 AND _bConnected THEN _intStep := _intStep + 10; END_IF
_w7 := _w6 AND NOT _bConnected;
IF _w7 THEN _intStep := _intFINAL_STEP; END_IF
IF _w7 THEN M_LogMessage(strMessage := 'Device not connected.'); END_IF
IF _w5 AND in_pDevice^.P_bError THEN _intStep := _intERROR_STEP; END_IF

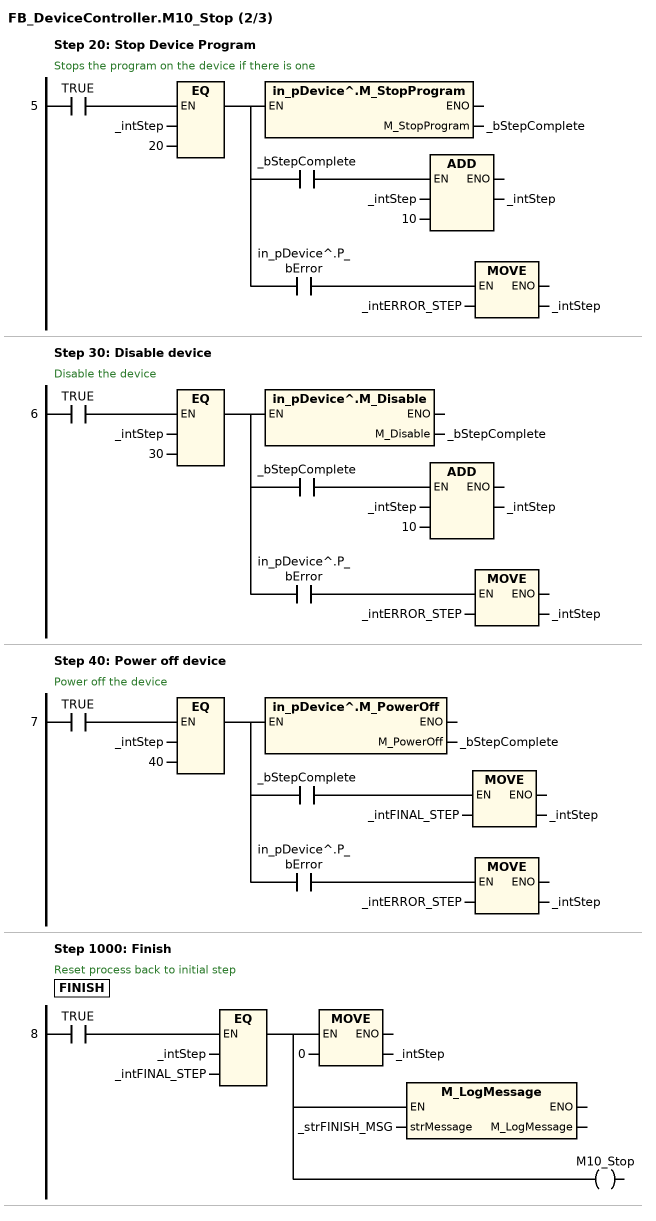
// NETWORK 5: Step 20: Stop Device Program
// Stops the program on the device if there is one
_w8 := _intStep = 20;
IF _w8 THEN _bStepComplete := in_pDevice^.M_StopProgram(); END_IF
IF _w8 AND _bStepComplete THEN _intStep := _intStep + 10; END_IF
IF _w8 AND in_pDevice^.P_bError THEN _intStep := _intERROR_STEP; END_IF

// NETWORK 6: Step 30: Disable device
// Disable the device
_w9 := _intStep = 30;
IF _w9 THEN _bStepComplete := in_pDevice^.M_Disable(); END_IF
IF _w9 AND _bStepComplete THEN _intStep := _intStep + 10; END_IF
IF _w9 AND in_pDevice^.P_bError THEN _intStep := _intERROR_STEP; END_IF

// NETWORK 7: Step 40: Power off device
// Power off the device
_w10 := _intStep = 40;
IF _w10 THEN _bStepComplete := in_pDevice^.M_PowerOff(); END_IF
IF _w10 AND _bStepComplete THEN _intStep := _intFINAL_STEP; END_IF
IF _w10 AND in_pDevice^.P_bError THEN _intStep := _intERROR_STEP; END_IF

// NETWORK 8: Step 1000: Finish
// Reset process back to initial step
FINISH:
_w11 := _intStep = _intFINAL_STEP;
IF _w11 THEN _intStep := 0; END_IF
IF _w11 THEN M_LogMessage(strMessage := _strFINISH_MSG); END_IF
M10_Stop := _w11;

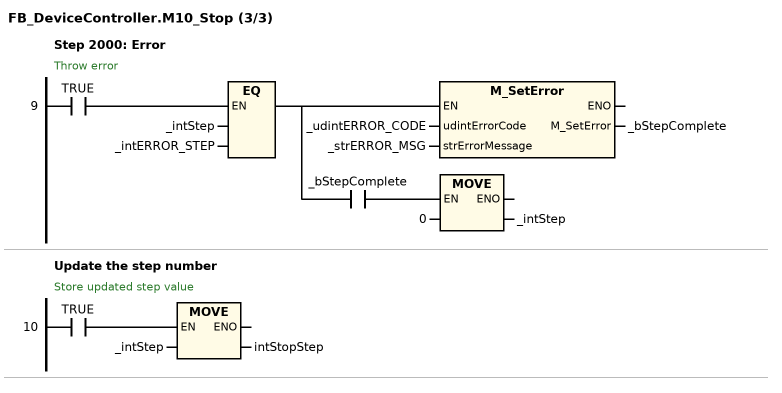
// NETWORK 9: Step 2000: Error
// Throw error
_w12 := _intStep = _intERROR_STEP;
IF _w12 THEN
    _bStepComplete := M_SetError(udintErrorCode := _udintERROR_CODE, strErrorMessage := _strERROR_MSG);
END_IF
IF _w12 AND _bStepComplete THEN _intStep := 0; END_IF

// NETWORK 10: Update the step number
// Store updated step value
intStopStep := _intStep;
END_METHOD

(* Connects, resets, and powers on the device. *)
METHOD M20_Reset : BOOL
VAR CONSTANT
	_intFINAL_STEP : INT := 1000;
	_intERROR_STEP : INT := 2000;
	_udintERROR_CODE: UDINT := E_DeviceControllerError.ResetError;
	_strERROR_MSG: T_MaxString := 'Error while trying to reset device!';
	_strSTART_MSG: T_MaxString := 'Resetting device';
	_strFINISH_MSG: T_MaxString := 'Device reset';
END_VAR
VAR
	_bStepComplete: BOOL;
	_intStep: INT;
END_VAR
VAR_INST // added by the converter: edge detectors and wires of the graphical bodies
    _w1, _w2, _w3, _w4, _w5, _w6, _w7, _w8, _w9 : BOOL;
END_VAR
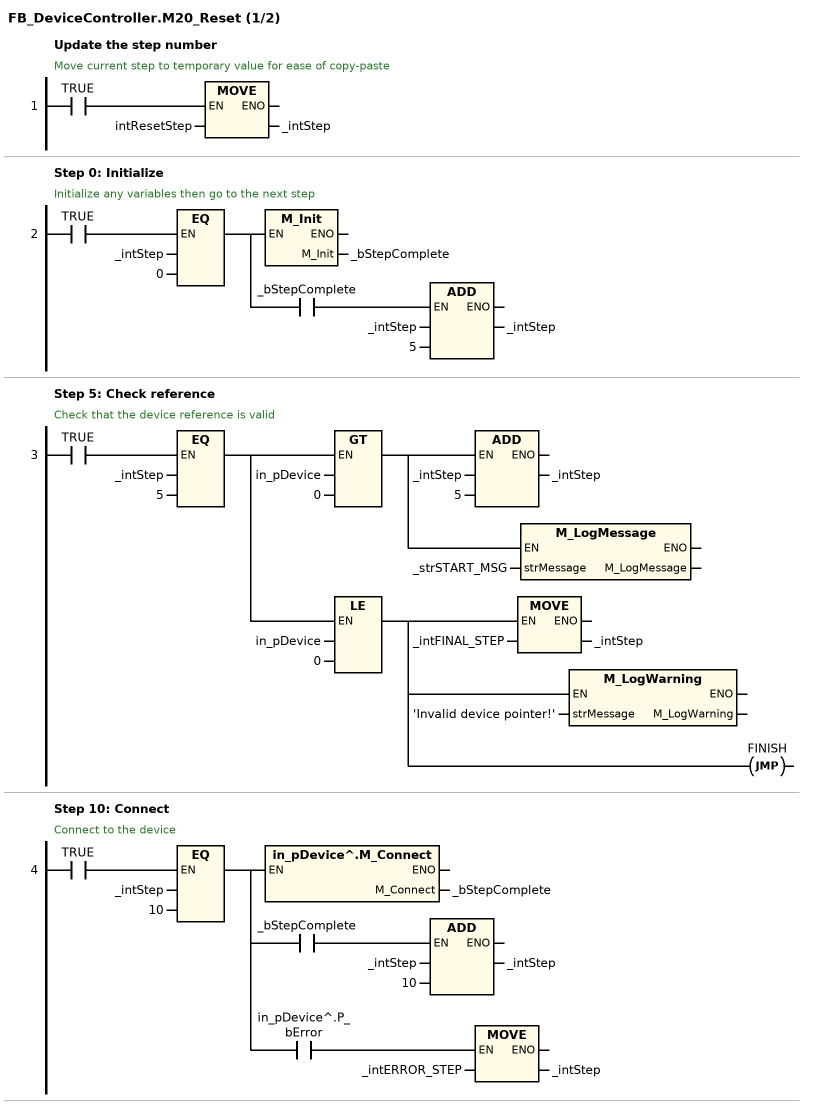
// NETWORK 1: Update the step number
// Move current step to temporary value for ease of copy-paste
_intStep := intResetStep;

// NETWORK 2: Step 0: Initialize
// Initialize any variables then go to the next step
_w1 := _intStep = 0;
IF _w1 THEN _bStepComplete := M_Init(); END_IF
IF _w1 AND _bStepComplete THEN _intStep := _intStep + 5; END_IF

// NETWORK 3: Step 5: Check reference
// Check that the device reference is valid
_w2 := _intStep = 5;
_w3 := _w2 AND in_pDevice > 0;
IF _w3 THEN _intStep := _intStep + 5; END_IF
IF _w3 THEN M_LogMessage(strMessage := _strSTART_MSG); END_IF
_w4 := _w2 AND in_pDevice <= 0;
IF _w4 THEN _intStep := _intFINAL_STEP; END_IF
IF _w4 THEN M_LogWarning(strMessage := 'Invalid device pointer!'); END_IF
IF _w4 THEN JMP FINISH; END_IF

// NETWORK 4: Step 10: Connect
// Connect to the device
_w5 := _intStep = 10;
IF _w5 THEN _bStepComplete := in_pDevice^.M_Connect(); END_IF
IF _w5 AND _bStepComplete THEN _intStep := _intStep + 10; END_IF
IF _w5 AND in_pDevice^.P_bError THEN _intStep := _intERROR_STEP; END_IF

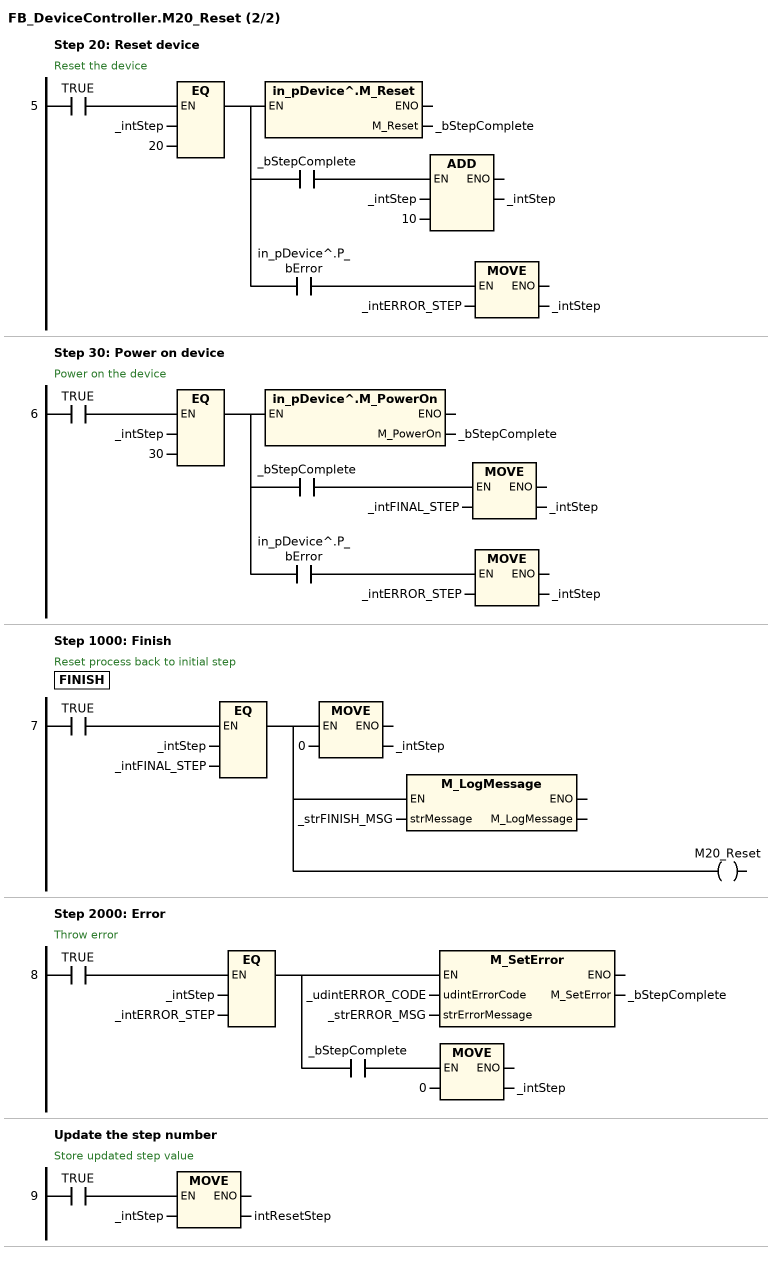
// NETWORK 5: Step 20: Reset device
// Reset the device
_w6 := _intStep = 20;
IF _w6 THEN _bStepComplete := in_pDevice^.M_Reset(); END_IF
IF _w6 AND _bStepComplete THEN _intStep := _intStep + 10; END_IF
IF _w6 AND in_pDevice^.P_bError THEN _intStep := _intERROR_STEP; END_IF

// NETWORK 6: Step 30: Power on device
// Power on the device
_w7 := _intStep = 30;
IF _w7 THEN _bStepComplete := in_pDevice^.M_PowerOn(); END_IF
IF _w7 AND _bStepComplete THEN _intStep := _intFINAL_STEP; END_IF
IF _w7 AND in_pDevice^.P_bError THEN _intStep := _intERROR_STEP; END_IF

// NETWORK 7: Step 1000: Finish
// Reset process back to initial step
FINISH:
_w8 := _intStep = _intFINAL_STEP;
IF _w8 THEN _intStep := 0; END_IF
IF _w8 THEN M_LogMessage(strMessage := _strFINISH_MSG); END_IF
M20_Reset := _w8;

// NETWORK 8: Step 2000: Error
// Throw error
_w9 := _intStep = _intERROR_STEP;
IF _w9 THEN
    _bStepComplete := M_SetError(udintErrorCode := _udintERROR_CODE, strErrorMessage := _strERROR_MSG);
END_IF
IF _w9 AND _bStepComplete THEN _intStep := 0; END_IF

// NETWORK 9: Update the step number
// Store updated step value
intResetStep := _intStep;
END_METHOD

(* Loads program and starts device then returns TRUE. *)
METHOD M30_Start : BOOL
VAR CONSTANT
	_udintERROR_CODE: UDINT := E_DeviceControllerError.StartError;
	_strERROR_MSG: T_MaxString := 'Error while trying to start device!';
	_intFINAL_STEP : INT := 1000;
	_intERROR_STEP : INT := 2000;
	_strSTART_MSG: T_MaxString := 'Starting device';
	_strFINISH_MSG: T_MaxString := 'Device started';
END_VAR
VAR
	_bStepComplete: BOOL;
	_intStep: INT;
END_VAR
VAR_INST // added by the converter: edge detectors and wires of the graphical bodies
    _w1, _w2, _w3, _w4, _w5, _w6, _w7, _w8, _w9 : BOOL;
END_VAR
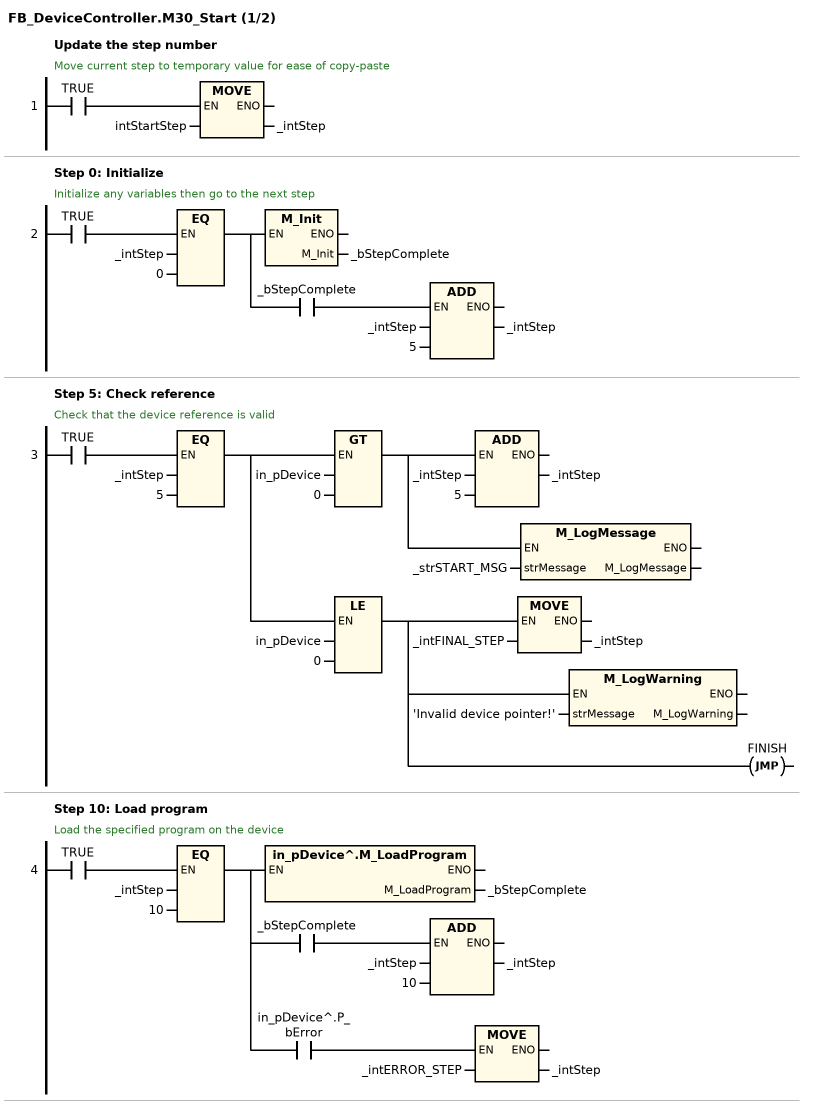
// NETWORK 1: Update the step number
// Move current step to temporary value for ease of copy-paste
_intStep := intStartStep;

// NETWORK 2: Step 0: Initialize
// Initialize any variables then go to the next step
_w1 := _intStep = 0;
IF _w1 THEN _bStepComplete := M_Init(); END_IF
IF _w1 AND _bStepComplete THEN _intStep := _intStep + 5; END_IF

// NETWORK 3: Step 5: Check reference
// Check that the device reference is valid
_w2 := _intStep = 5;
_w3 := _w2 AND in_pDevice > 0;
IF _w3 THEN _intStep := _intStep + 5; END_IF
IF _w3 THEN M_LogMessage(strMessage := _strSTART_MSG); END_IF
_w4 := _w2 AND in_pDevice <= 0;
IF _w4 THEN _intStep := _intFINAL_STEP; END_IF
IF _w4 THEN M_LogWarning(strMessage := 'Invalid device pointer!'); END_IF
IF _w4 THEN JMP FINISH; END_IF

// NETWORK 4: Step 10: Load program
// Load the specified program on the device
_w5 := _intStep = 10;
IF _w5 THEN _bStepComplete := in_pDevice^.M_LoadProgram(); END_IF
IF _w5 AND _bStepComplete THEN _intStep := _intStep + 10; END_IF
IF _w5 AND in_pDevice^.P_bError THEN _intStep := _intERROR_STEP; END_IF

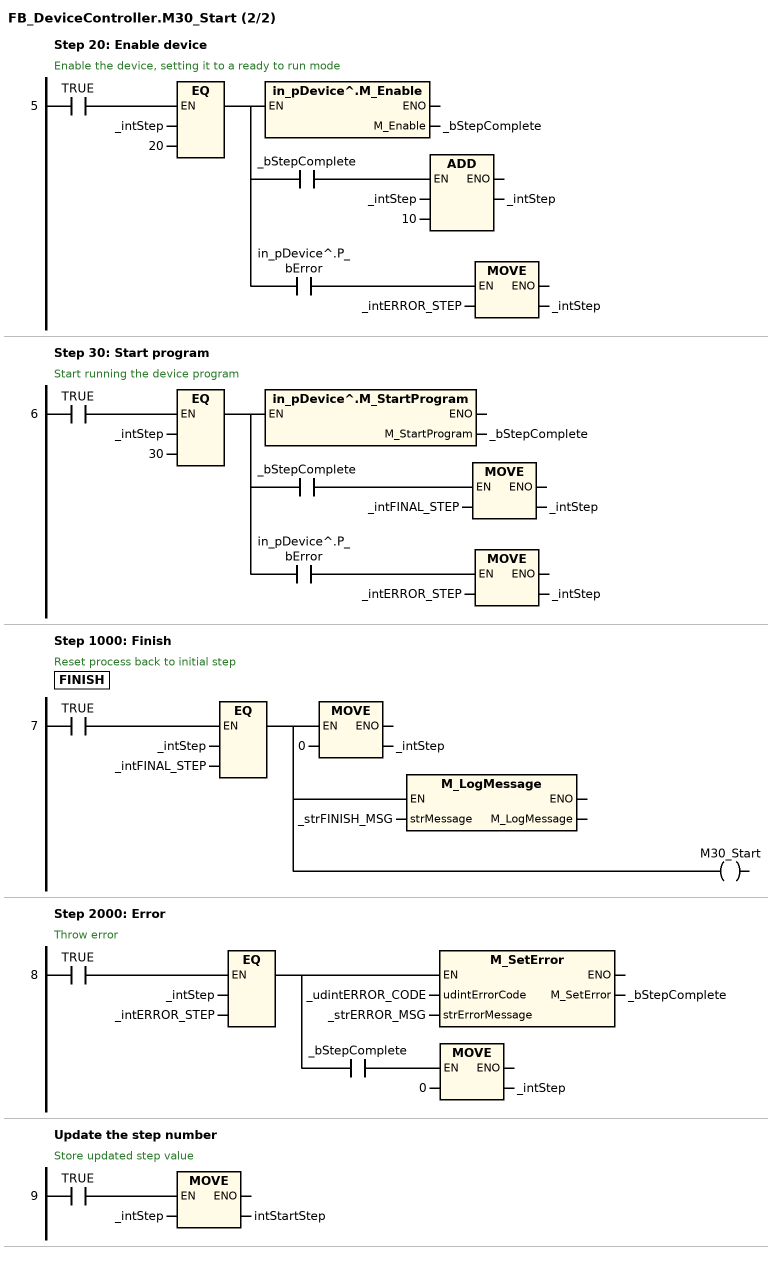
// NETWORK 5: Step 20: Enable device
// Enable the device, setting it to a ready to run mode
_w6 := _intStep = 20;
IF _w6 THEN _bStepComplete := in_pDevice^.M_Enable(); END_IF
IF _w6 AND _bStepComplete THEN _intStep := _intStep + 10; END_IF
IF _w6 AND in_pDevice^.P_bError THEN _intStep := _intERROR_STEP; END_IF

// NETWORK 6: Step 30: Start program
// Start running the device program
_w7 := _intStep = 30;
IF _w7 THEN _bStepComplete := in_pDevice^.M_StartProgram(); END_IF
IF _w7 AND _bStepComplete THEN _intStep := _intFINAL_STEP; END_IF
IF _w7 AND in_pDevice^.P_bError THEN _intStep := _intERROR_STEP; END_IF

// NETWORK 7: Step 1000: Finish
// Reset process back to initial step
FINISH:
_w8 := _intStep = _intFINAL_STEP;
IF _w8 THEN _intStep := 0; END_IF
IF _w8 THEN M_LogMessage(strMessage := _strFINISH_MSG); END_IF
M30_Start := _w8;

// NETWORK 8: Step 2000: Error
// Throw error
_w9 := _intStep = _intERROR_STEP;
IF _w9 THEN
    _bStepComplete := M_SetError(udintErrorCode := _udintERROR_CODE, strErrorMessage := _strERROR_MSG);
END_IF
IF _w9 AND _bStepComplete THEN _intStep := 0; END_IF

// NETWORK 9: Update the step number
// Store updated step value
intStartStep := _intStep;
END_METHOD

(* Stops and disables the device then returns TRUE when done. *)
METHOD M32_Complete : BOOL
VAR CONSTANT
	_udintERROR_CODE: UDINT := E_DeviceControllerError.CompleteError;
	_strERROR_MSG: T_MaxString := 'Error while trying to complete device!';
	_intFINAL_STEP : INT := 1000;
	_intERROR_STEP : INT := 2000;
	_strSTART_MSG: T_MaxString := 'Completing device';
	_strFINISH_MSG: T_MaxString := 'Device completed';
END_VAR
VAR
	_bStepComplete: BOOL;
	_intStep: INT;
END_VAR
VAR_INST // added by the converter: edge detectors and wires of the graphical bodies
    _w1, _w2, _w3, _w4, _w5, _w6, _w7, _w8 : BOOL;
END_VAR
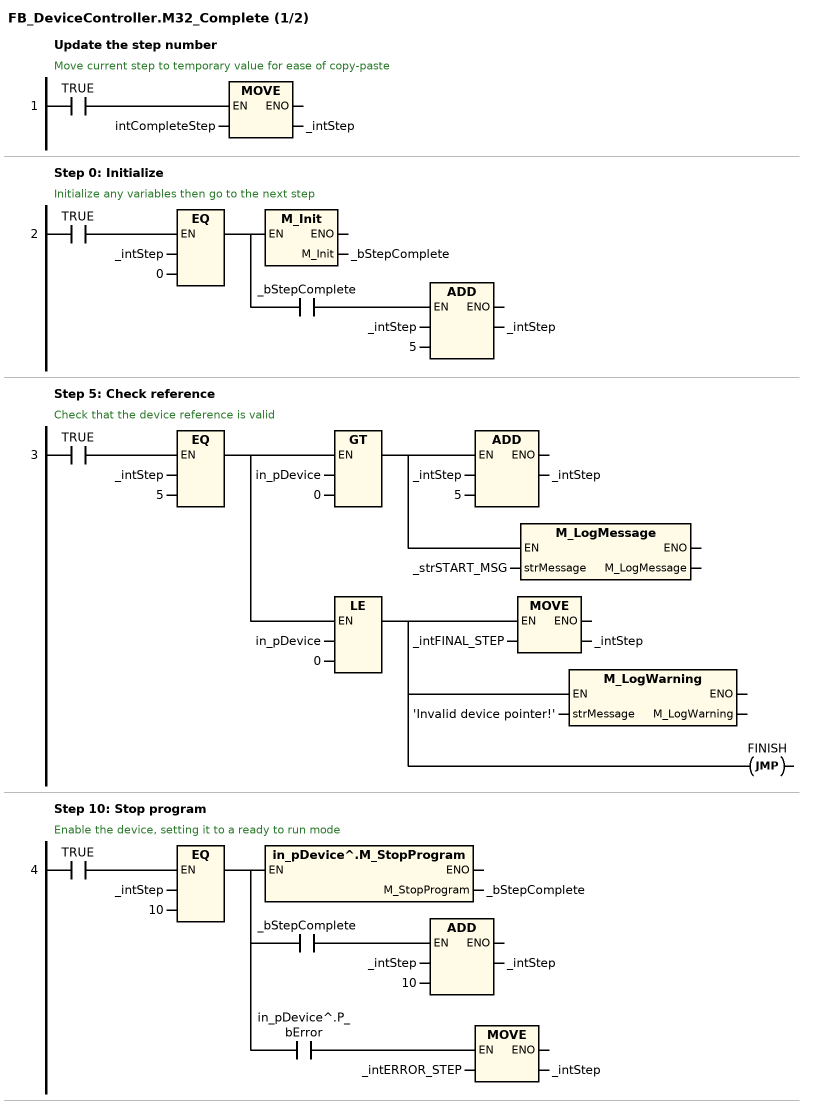
// NETWORK 1: Update the step number
// Move current step to temporary value for ease of copy-paste
_intStep := intCompleteStep;

// NETWORK 2: Step 0: Initialize
// Initialize any variables then go to the next step
_w1 := _intStep = 0;
IF _w1 THEN _bStepComplete := M_Init(); END_IF
IF _w1 AND _bStepComplete THEN _intStep := _intStep + 5; END_IF

// NETWORK 3: Step 5: Check reference
// Check that the device reference is valid
_w2 := _intStep = 5;
_w3 := _w2 AND in_pDevice > 0;
IF _w3 THEN _intStep := _intStep + 5; END_IF
IF _w3 THEN M_LogMessage(strMessage := _strSTART_MSG); END_IF
_w4 := _w2 AND in_pDevice <= 0;
IF _w4 THEN _intStep := _intFINAL_STEP; END_IF
IF _w4 THEN M_LogWarning(strMessage := 'Invalid device pointer!'); END_IF
IF _w4 THEN JMP FINISH; END_IF

// NETWORK 4: Step 10: Stop program
// Enable the device, setting it to a ready to run mode
_w5 := _intStep = 10;
IF _w5 THEN _bStepComplete := in_pDevice^.M_StopProgram(); END_IF
IF _w5 AND _bStepComplete THEN _intStep := _intStep + 10; END_IF
IF _w5 AND in_pDevice^.P_bError THEN _intStep := _intERROR_STEP; END_IF

